# B&R Automation Studio project NAEUL004C00R13L518F00 (part 11)

#### Act_OptPage.st
```iecst
ACTION Act_OptPage:

	//Prevent Screen Saver Interupt Program
	IF tyProperty.tyVisu.uiCurrPage <> 0 THEN
		eCurrPage := tyProperty.tyVisu.uiCurrPage;
	ELSE
		Act_OptP0000McStatus;
		Act_OptP0000RunningNm;
		Act_OptP0000StatDisp;
	END_IF

	Act_OptP0000DisableSSaver;
	Act_OptP0000TouchTimer;			//Auto Logout
	Act_OptP0000Hermes; 	//Changed

	IF (tyProperty.tyVisu.uiChgPage = 65535) AND (usiChgPage = 0) THEN

		Act_OptC0005GoHomeCtrl;
		Act_OptC0005ShowNotif;
		Act_OptC0005AutoCtrl;
		Act_OptC0005RstErr;
		Act_OptC0005StatBarCtrl;
		Act_OptC0005Buzzer;
		Act_OptC0005ChgPage;
		Act_OptC0007Notif;
		Act_OptC0009Info;

		Act_OptP0202InsertRmvMag;
		Act_OptP0203InsertRmvMag;
		Act_OptP0204InsertRmvMag;

		CASE eCurrPage OF

			UIP0001Startup:
				Act_OptP0001Startup;

			UIP0100Login:
				Act_OptP0100Keypad;
				Act_OptP0100NomLogin;
				Act_OptP0100BypassLogin;
				Act_OptP0100Logout;

			UIP0200OpsGen:
				Act_OptP0200ChgPage;
				Act_OptP0200UpdtDat;
				Act_OptP0200VSMEMA;
				Act_OptP0200RcyMsg;
				Act_OptP0200ToP0204_P0003AccDat;
				Act_OptP0200ToP0204BypsInitConv;
				Act_OptP0202RstMnl;
				Act_OptP0203RstMnl;
				Act_OptP0204RstMnl;

			UIP0201OpsTravLifter:
				Act_OptP0201Navi;
				Act_OptP0201UpdtDat;
				Act_OptP0201IOMonitor;
				Act_OptP0201ChgParam;
				Act_OptP0200ToP0204_P0003AccDat;
				Act_OptP0200ToP0204BypsInitConv;
					//Changed
				Act_OptP0201QueryBoardInfo;
				Act_OptP0201CurrWorkOrderInfo;
				Act_OptP0201QueryWorkOrderInfo;
				Act_OptP0201BarcodeScanner;

			UIP0202OpsMag1:
				Act_OptP0202Navi;
				Act_OptP0202UpdtDat;
				Act_OptP0202IOMonitor;
				Act_OptP0202ChgPage;
				Act_OptP0202_P0003AIVDat;
				Act_OptP0202ChgParam;
				Act_OptP0200ToP0204_P0003AccDat;
				Act_OptP0200ToP0204BypsInitConv;
				Act_OptP0202ToP0204_P0003UnloadMag;
				IF p_tyNtParamCurr.bProjMagConvLane1Prep THEN
					Act_OptP0202Lane1ChgMag;
				END_IF
			UIP0203OpsMag2:
				Act_OptP0203Navi;
				Act_OptP0203UpdtDat;
				Act_OptP0203IOMonitor;
				Act_OptP0203ChgPage;
				Act_OptP0203_P0003AIVDat;
				Act_OptP0203ChgParam;
				Act_OptP0200ToP0204_P0003AccDat;
				Act_OptP0200ToP0204BypsInitConv;
				Act_OptP0202ToP0204_P0003UnloadMag;
				IF p_tyNtParamCurr.bProjMagConvLane2Prep THEN
					Act_OptP0203Lane2ChgMag;
				END_IF
			UIP0204OpsMag3:
				Act_OptP0204Navi;
				Act_OptP0204UpdtDat;
				Act_OptP0204IOMonitor;
				Act_OptP0204ChgPage;
				Act_OptP0204_P0003AIVDat;
				Act_OptP0204ChgParam;
				Act_OptP0200ToP0204_P0003AccDat;
				Act_OptP0200ToP0204BypsInitConv;
				Act_OptP0202ToP0204_P0003UnloadMag;

			UIP0205OpsAIV:
				Act_OptP0205Navi;
				Act_OptP0205IOMonitor;

			UIP0206OpsMagConv1:
				Act_OptP0206Navi;
				Act_OptP0206UpdtDat;
				Act_OptP0206IOMonitor;
				Act_OptP0200ToP0204_P0003AccDat;
				Act_OptP0200ToP0204BypsInitConv;

			UIP0207OpsMagConv2:
				Act_OptP0207Navi;
				Act_OptP0207UpdtDat;
				Act_OptP0207IOMonitor;
				Act_OptP0200ToP0204_P0003AccDat;
				Act_OptP0200ToP0204BypsInitConv;

			UIP0300McInfo:

			UIP0400ProdSel:
				Act_OptP0400Search;
				Act_OptP0400Load;
				Act_OptP0400Preview;
				Act_OptP0400Table;
				Act_OptP0400Keypad;
				Act_OptP0400Mask;
				Act_OptP0400Sort;
				Act_OptP0400RcpPopUp;

			UIP0410MagSel:
				Act_OptP0410Load;
				Act_OptP0410Preview;
				Act_OptP0410Table;
				Act_OptP0410Mask;
				Act_OptP0410Sort;

			UIP0600Alm:
				Act_OptP0600Alm;
				Act_OptP0600RcyMsg;

			UIP0700LFCtrl:
				Act_OptP0700LFLeaderCtrl;
				Act_OptP0700Mask;
				Act_OptP0700Table;

			UIP0800MagInfo:
				Act_OptP0800Table1;
				Act_OptP0800Mag1Updt;
				Act_OptP0800Table2;
				Act_OptP0800Mag2Updt;
				Act_OptP0800Table3;
				Act_OptP0800Mag3Updt;

			UIP0850OvenInfo:
				Act_OptP0850UpdtDat;
				Act_OptP0850BrdInOven;
				Act_OptP0850Keypad;

				UIP0002Menu,UIP0003MMenu, UIP0900GenIn, UIP0910GenOut, UIP0920MtrNPneuCtrl, UIP0921Shutter, UIP0922Stopper, UIP0923SafetyBar, UIP0926LifterConv, UIP0927LifterConv2, UIP0928MagConv, UIP0929MagConv2,UIP0930MagConv1, UIP0931MagConv2, UIP0932MagConv3, UIP0933PusherConv,
				 UIP0934AW, UIP0935Lifter, UIP0936Trav, UIP0937AWPushOrPuller, UIP0938MagAW, UIP0939Lifter2,UIP0940CommCtrl:
				IF eCurrPage = UIP0002Menu THEN
					Act_OptP0002Mask;
					Act_OptP0002ChgPage;
					Act_OptP0002MsgGuide;
					Act_OptP0002UpdtData;
				END_IF

				IF eCurrPage = UIP0003MMenu THEN
					Act_OptP0003UpdtStat;
					Act_OptP0202ToP0204_P0003UnloadMag;
					Act_OptP0200ToP0204_P0003AccDat;
					Act_OptP0202_P0003AIVDat;
					Act_OptP0203_P0003AIVDat;
					Act_OptP0204_P0003AIVDat;
				END_IF

				Act_OptP0002ManualCtrl;
				Act_OptP0910RstMnl;
				Act_OptP0921RstMnl;
				Act_OptP0922RstMnl;
				Act_OptP0923RstMnl;
				IF p_tyNtParamCurr.bProjMagConvLane1Prep THEN
					Act_OptP0926RstMnl;
					Act_OptP0928RstMnlTop;
					Act_OptP0928RstMnlBtm;
				END_IF
				IF p_tyNtParamCurr.bProjMagConvLane2Prep THEN
					Act_OptP0927RstMnl;
					Act_OptP0929RstMnlTop;
					Act_OptP0929RstMnlBtm;
				END_IF
				Act_OptP0930RstMnl;
				Act_OptP0931RstMnl;
				Act_OptP0932RstMnl;
				Act_OptP0933RstMnl;
				Act_OptP0934RstMnl;
				Act_OptP0935RstMnl;
				Act_OptP0936RstMnl;
				Act_OptP0937RstMnl;
				Act_OptP0938RstMnl;
				IF p_tyNtParamCurr.bProjLifter2Prep THEN
					Act_OptP0939RstMnl;
				END_IF
				Act_OptP0940RstMnl;
				Act_OptP0950RstMnl;
				Act_OptP0202RstMnl;
				Act_OptP0203RstMnl;
				Act_OptP0204RstMnl;
				Act_OptP0205RstMnl;

				IF bUIManualMod = TRUE THEN

					//General Input
					Act_OptP0900ReadDI;

					//General Output
					Act_OptP0910WriteDO;

					//MtrNPneuCtrl
					Act_OptP0920FullMask;
					Act_OptP0920ChgPage;

					//Inlet & Outlet Shutter
					Act_OptP0921DualMask;
					Act_OptP0921Navi;
					Act_OptP0921InletShutterChgLyr;
					Act_OptP0921InletShutterSen;
					Act_OptP0921InletShutterFB;
					Act_OptP0921InletShutterFBStat;
					Act_OptP0921InletShutterDC;
					Act_OptP0921OutletShutterChgLyr;
					Act_OptP0921OutletShutterSen;
					Act_OptP0921OutletShutterFB;
					Act_OptP0921OutletShutterFBStat;
					Act_OptP0921OutletShutterDC;
					Act_OptP0921OutletShutterChgLyr2;
					Act_OptP0921OutletShutterSen2;
					Act_OptP0921OutletShutterFB2;
					Act_OptP0921OutletShutterFBStat2;
					Act_OptP0921OutletShutterDC2;
					Act_OptP0921OutletShutterChgLyr3;
					Act_OptP0921OutletShutterSen3;
					Act_OptP0921OutletShutterFB3;
					Act_OptP0921OutletShutterFBStat3;
					Act_OptP0921OutletShutterDC3;

					//Stopper A & B
					Act_OptP0922DualMask;
					Act_OptP0922Navi;
					Act_OptP0922StopperAChgLyr;
					Act_OptP0922StopperASen;
					Act_OptP0922StopperAFB;
					Act_OptP0922StopperAFBStat;
					Act_OptP0922StopperADC;
					Act_OptP0922StopperBChgLyr;
					Act_OptP0922StopperBSen;
					Act_OptP0922StopperBFB;
					Act_OptP0922StopperBFBStat;
					Act_OptP0922StopperBDC;
					Act_OptP0922InStopperChgLyr;
					Act_OptP0922InStopperSen;
					Act_OptP0922InStopperFB;
					Act_OptP0922InStopperFBStat;
					Act_OptP0922InStopperDC;

					//Safety Bar
					Act_OptP0923DualMask;
					Act_OptP0923Navi;
					Act_OptP0923Mag1SafetyBarChgLyr;
					Act_OptP0923Mag1SafetyBarSen;
					Act_OptP0923Mag1SafetyBarFB;
					Act_OptP0923Mag1SafetyBarFBStat;
					Act_OptP0923Mag1SafetyBarDC;
					Act_OptP0923Mag2SafetyBarChgLyr;
					Act_OptP0923Mag2SafetyBarSen;
					Act_OptP0923Mag2SafetyBarFB;
					Act_OptP0923Mag2SafetyBarFBStat;
					Act_OptP0923Mag2SafetyBarDC;
					Act_OptP0923Mag3SafetyBarChgLyr;
					Act_OptP0923Mag3SafetyBarSen;
					Act_OptP0923Mag3SafetyBarFB;
					Act_OptP0923Mag3SafetyBarFBStat;
					Act_OptP0923Mag3SafetyBarDC;

					IF p_tyNtParamCurr.bProjMagConvLane1Prep  THEN
						//Lifter Magazine Conveyor
						Act_OptP0926FullMask;
						Act_OptP0926Navi;
						Act_OptP0926LifterMagConvChgLyr;
						Act_OptP0926LifterMagConvSen;
						Act_OptP0926LifterMagConvFB;
						Act_OptP0926LifterMagConvFBStat;
						Act_OptP0926LifterMagConvDC;

						//MagConv Lane1
						Act_OptP0928FullMask;
						Act_OptP0928Navi;
						Act_OptP0928MagConv1ChgLyr;
						Act_OptP0928MagConv1Sen;
						Act_OptP0928MagConv1TopFB;
						Act_OptP0928MagConv1BtmFB;
						Act_OptP0928MagConv1FBStat;
						Act_OptP0928MagConv1TopDC;
						Act_OptP0928MagConv1BtmDC;
					END_IF

					IF p_tyNtParamCurr.bProjMagConvLane2Prep  THEN
						//Lifter Magazine Conveyor2
						Act_OptP0927FullMask;
						Act_OptP0927Navi;
						Act_OptP0927LifterMagConvChgLyr;
						Act_OptP0927LifterMagConvSen;
						Act_OptP0927LifterMagConvFB;
						Act_OptP0927LifterMagConvFBStat;
						Act_OptP0927LifterMagConvDC;

						//MagConv Lane2
						Act_OptP0929FullMask;
						Act_OptP0929Navi;
						Act_OptP0929MagConv2ChgLyr;
						Act_OptP0929MagConv2Sen;
						Act_OptP0929MagConv2TopFB;
						Act_OptP0929MagConv2BtmFB;
						Act_OptP0929MagConv2FBStat;
						Act_OptP0929MagConv2TopDC;
						Act_OptP0929MagConv2BtmDC;
					END_IF

					//Magazine Conveyor 1
					Act_OptP0930FullMask;
					Act_OptP0930Navi;
					Act_OptP0930MagConv1ChgLyr;
					Act_OptP0930MagConv1Sen;
					Act_OptP0930MagConv1FB;
					Act_OptP0930MagConv1FBStat;
					Act_OptP0930MagConv1DC;

					//Magazine Conveyor 2
					Act_OptP0931FullMask;
					Act_OptP0931Navi;
					Act_OptP0931MagConv2ChgLyr;
					Act_OptP0931MagConv2Sen;
					Act_OptP0931MagConv2FB;
					Act_OptP0931MagConv2FBStat;
					Act_OptP0931MagConv2DC;

					//Magazine Conveyor 3
					Act_OptP0932FullMask;
					Act_OptP0932Navi;
					Act_OptP0932MagConv3ChgLyr;
					Act_OptP0932MagConv3Sen;
					Act_OptP0932MagConv3FB;
					Act_OptP0932MagConv3FBStat;
					Act_OptP0932MagConv3DC;

					//Pusher Conveyor
					Act_OptP0933FullMask;
					Act_OptP0933Navi;
					Act_OptP0933PusherConvChgLyr;
					Act_OptP0933PusherConvSen;
					Act_OptP0933PusherConvFB;
					Act_OptP0933PusherConvFBStat;
					Act_OptP0933PusherConvDC;

					//AutoWidth
					Act_OptP0934FullMask;
					Act_OptP0934Navi;
					Act_OptP0934FBCtrl;
					Act_OptP0934FBStat;
					Act_OptP0934Mask;
					Act_OptP0934UpdtDat;
					Act_OptP0934Keypad;

					//Lifter
					Act_OptP0935FullMask;
					Act_OptP0935Navi;
					Act_OptP0935FBCtrl;
					Act_OptP0935FBStat;
					Act_OptP0935Mask;
					Act_OptP0935UpdtDat;
					Act_OptP0935Keypad;

					//Traverser
					Act_OptP0936FullMask;
					Act_OptP0936Navi;
					Act_OptP0936FBCtrl;
					Act_OptP0936FBStat;
					Act_OptP0936Mask;
					Act_OptP0936UpdtDat;
					Act_OptP0936Keypad;

					//Pusher Or Puller Auto Width
					Act_OptP0937FullMask;
					Act_OptP0937Navi;
					Act_OptP0937FBCtrl;
					Act_OptP0937FBStat;
					Act_OptP0937Mask;
					Act_OptP0937UpdtDat;
					Act_OptP0937Keypad;

					//Magazine Auto Width
					Act_OptP0938FullMask;
					Act_OptP0938Navi;
					Act_OptP0938FBCtrl1;
					Act_OptP0938FBCtrl2;
					Act_OptP0938FBCtrl3;
					Act_OptP0938FBStat;
					Act_OptP0938Mask;
					Act_OptP0938UpdtDat;
					Act_OptP0938Keypad;

					//Lifter 2
					IF p_tyNtParamCurr.bProjLifter2Prep THEN
						Act_OptP0939FullMask;
						Act_OptP0939Navi;
						Act_OptP0939FBCtrl;
						Act_OptP0939FBStat;
						Act_OptP0939Mask;
						Act_OptP0939UpdtDat;
						Act_OptP0939Keypad;
					END_IF
					//Communication
					Act_OptP0940FullMask;
					Act_OptP0940ReadDI;
					Act_OptP0940WriteDO;

				END_IF

			UIP0950Simu:
				Act_OptP0950Navi;
				Act_OptP0950Ctrl;
				Act_OptP0950SimuMod;
				//Act_OptP0950DispBffrCycle;

			UIP1000Lang:
				Act_OptP1000SelectLang;
				Act_OptP1000Keypad;

			UIP1020McSetNavi:
				Act_OptP1020Navi;

			UIP1021McSetGen:
				Act_OptP1021Navi;
				Act_OptP1021Save;
				Act_OptP1021Keypad;
				Act_OptP1021Teach;
				Act_OptP1021IPAddr;
				Act_OptP1021SubnetMask;
				Act_OptP1021HMIIPAddr;
				Act_OptP1021DHCPSetting;

			UIP1022McSetVComm:
				Act_OptP1022Navi;
				Act_OptP1022Save;
				Act_OptP1022DisLF;
				Act_OptP1022Keypad; //new for Hermes 1.3

			UIP1023McSetHComm:
				Act_OptP1023Navi;
				Act_OptP1023ShowLyr;
				Act_OptP1023Save;
				Act_OptP1023USSel;
				Act_OptP1023Keypad;

			UIP1024McSetAntiGap:
				Act_OptP1024Navi;
				Act_OptP1024Save;
				Act_OptP1024Keypad;

			UIP1025McSetScan:
				Act_OptP1025Navi;
				Act_OptP1025Save;
				Act_OptP1025Keypad;

			UIP1026McSetTeach:
				Act_OptP1026Navi;
				Act_OptP1026FullMask;
				Act_OptP1026Mnl;

				//Traverser
				Act_OptP1026TravTeach;
				Act_OptP1026TravFBCtrl;
				Act_OptP1026TravFBStat;
				Act_OptP1026TravMask;
				Act_OptP1026TravUpdtDat;
				Act_OptP1026TravKeypad;
				Act_OptP1026TravRstMnl;

				//Lifter
				Act_OptP1026LifterTeach;
				IF (bTeachLifterTopPos2 OR bTeachLifterBtmPos2) AND  p_tyNtParamCurr.bProjLifter2Prep THEN
					Act_OptP1026Lifter2FBCtrl;
					Act_OptP1026Lifter2FBStat;
					Act_OptP1026Lifter2Mask;
					Act_OptP1026Lifter2UpdtDat;
				ELSE
					Act_OptP1026LifterFBCtrl;
					Act_OptP1026LifterFBStat;
					Act_OptP1026LifterMask;
					Act_OptP1026LifterUpdtDat;
				END_IF
				Act_OptP1026LifterKeypad;
				Act_OptP1026LifterRstMnl;

			UIP1027McSetOpCon:
				Act_OptP1027Navi;
				Act_OptP1027Save;
				Act_OptP1027Keypad;

			UIP1030MagSet:
				Act_OptP1030Mask;
				Act_OptP1030Save;
				Act_OptP1030Del;
				Act_OptP1030Table;
				Act_OptP1030LoadData;
				Act_OptP1030Keypad;
				Act_OptP1030Teach;
				Act_OptP1030Sort;

			UIP1031MagSetTeach:
				Act_OptP1031Navi;
				Act_OptP1031FullMask;
				Act_OptP1031Mnl;

				//Traverser
				Act_OptP1031TravTeach;
				Act_OptP1031TravFBCtrl;
				Act_OptP1031TravFBStat;
				Act_OptP1031TravMask;
				Act_OptP1031TravUpdtDat;
				Act_OptP1031TravKeypad;
				Act_OptP1031TravRstMnl;

				//Lifter
				Act_OptP1031LifterTeach;

				IF p_tyNtParamCurr.bProjMagConvLane2Prep AND bTeachLifterMag2Slt1Pos AND  p_tyNtParamCurr.bProjLifter2Prep THEN
					Act_OptP1031Lifter2FBCtrl;
					Act_OptP1031Lifter2FBStat;
					Act_OptP1031Lifter2Mask;
					Act_OptP1031Lifter2UpdtDat;
				ELSE
					Act_OptP1031LifterFBCtrl;
					Act_OptP1031LifterFBStat;
					Act_OptP1031LifterMask;
					Act_OptP1031LifterUpdtDat;
				END_IF
				Act_OptP1031LifterKeypad;
				Act_OptP1031LifterRstMnl;

			UIP1040ProdSet:
				Act_OptP1040Mask;
				Act_OptP1040Save;
				Act_OptP1040Limit;
				Act_OptP1040Del;
				Act_OptP1040Table;
				Act_OptP1040LoadData;
				Act_OptP1040Search;
				Act_OptP1040Keypad;
				Act_OptP1040ToXML;
				Act_OptP1040FromXML;
				Act_OptP1040Sort;
				Act_OptP1040RcpPopUp;

			UIP1050LFSet:
				Act_OptP1050Keypad;
				Act_OptP1050Edit;
				Act_OptP1050Online;
				Act_OptP1050Offline;
				Act_OptP1050Delete;
				Act_OptP1050ShftUp;
				Act_OptP1050ShftDwn;
				Act_OptP1050Mask;
				Act_OptP1050Table;
				Act_OptP1050Oven;

			UIP1080UsrMgmt:
				Act_OptP1080Keypad;
				Act_OptP1080AddUsr;
				Act_OptP1080DelUsr;
				Act_OptP1080EditUsr;
				Act_OptP1080EditAccess;
				Act_OptP1080Table;

			UIP1081UsrMgmtUsrAccessRgt:
				Act_OptP1081Navi;
				Act_OptP1081Save;
				Act_OptP1081Load;
				Act_OptP1081Keypad;

		END_CASE

	END_IF

END_ACTION
```

#### Act_OptC0005GoHomeCtrl.st
```iecst
ACTION Act_OptC0005GoHomeCtrl:

	//Control
	IF tyCommon.tyMain.tyBtnHome.bRtCompl = TRUE OR tyCommon.tyMain1.tyBtnHome.bRtCompl = TRUE THEN
		tyCommon.tyMain.tyBtnHome.bRtCompl	:= FALSE;
		tyCommon.tyMain1.tyBtnHome.bRtCompl := FALSE;
		eChgPage							:= UIP0002Menu;
	END_IF

	//Go Main
	IF tyCommon.tyMain.tyBtnGoMain.bRtCompl = TRUE THEN
		tyCommon.tyMain.tyBtnGoMain.bRtCompl := FALSE;
		eChgPage		:= UIP0003MMenu;
	END_IF

	//Mask
	IF tyP0100Login.tyLogin.tyBtnLogin.bRtCompl 					OR tyP0100Login.tyLogout.tyBtnLogout.bRtCompl
		OR tyP0400ProdSel.tyProdSel.tyBtnLoad.bRtCompl 				OR tyP0400ProdSel.tyProdSel.tyStringSearch.bRtCompl
		OR tyP0410MagSel.tyMagSel.tyBtnLoad.bRtCompl				OR tyP0800MagInfo.tyMagInfo1.tyBtnMag1SetFull.bRtCompl
		OR tyP0800MagInfo.tyMagInfo1.tyBtnMag2SetFull.bRtCompl		OR tyP0800MagInfo.tyMagInfo2.tyBtnMag3SetFull.bRtCompl
		OR tyP1030MagSet.tyMagSet.tyBtnDelete.bRtCompl				OR tyP1030MagSet.tyMagSet.tyBtnSave.bRtCompl
		OR tyP1040ProdSet.tyProdSet.tyBtnDelete.bRtCompl			OR tyP1040ProdSet.tyProdSet.tyBtnSave.bRtCompl
		OR tyP1040ProdSet.tyProdSet.tyBtnToXML.bRtCompl				OR tyP1040ProdSet.tyProdSet.tyBtnFromXML.bRtCompl
		OR tyP1050LFSet.tyLdr.tyBtnDelete.bRtCompl					OR tyP1050LFSet.tyLdr.tyBtnOnline.bRtCompl
		OR tyP1050LFSet.tyLdr.tyBtnOffline.bRtCompl					OR tyP1050LFSet.tyLdr.tyBtnShftUp.bRtCompl
		OR tyP1050LFSet.tyLdr.tyBtnShftDwn.bRtCompl					OR tyP1080UsrMgmt.tyUsrMgmt.tyBtnDeleteUsr.bRtCompl
		OR tyP1080UsrMgmt.tyUsrMgmt.tyBtnEditDetail.bRtCompl		OR tyP1080UsrMgmt.tyUsrMgmt.tyBtnNewUsr.bRtCompl
		OR tyCommon.tySet.tyBtnSave.bRtCompl						OR bTeachTravPosA
		OR bTeachTravPosB											OR bTeachTravPosMag1
		OR bTeachTravPosMag2										OR bTeachTravPosMag3
		OR bTeachLifterPosA											OR bTeachLifterPosB
		OR bTeachLifterMag1Slt1Pos									OR bTeachLifterMag2Slt1Pos
		OR bTeachLifterMag3Slt1Pos
		OR p_bSimuStatusRun
		THEN

		fUIInRtStatOff(ADR(tyCommon.tyMain.tyBtnHome.uiMaskRtStat));
		fUIInRtStatOff(ADR(tyCommon.tyMain1.tyBtnHome.uiMaskRtStat));

		fUIInRtStatOff(ADR(tyCommon.tyMain.tyBtnGoMain.uiMaskRtStat));

	ELSIF bUIManualMod THEN
		fUIInRtStatHide(ADR(tyCommon.tyMain.tyBtnHome.uiMaskRtStat));
		fUIInRtStatHide(ADR(tyCommon.tyMain1.tyBtnHome.uiMaskRtStat));

		fUIInRtStatHide(ADR(tyCommon.tyMain.tyBtnGoMain.uiMaskRtStat));
	ELSE
		fUIInRtStatHide(ADR(tyCommon.tyMain.tyBtnHome.uiMaskRtStat));
		fUIInRtStatHide(ADR(tyCommon.tyMain1.tyBtnHome.uiMaskRtStat));

		fUIInRtStatHide(ADR(tyCommon.tyMain.tyBtnGoMain.uiMaskRtStat));
	END_IF

END_ACTION
```

#### Act_OptC0005ShowNotif.st
```iecst
ACTION Act_OptC0005ShowNotif:

	//Control
	IF tyCommon.tyMain.tyBtnNotification.bRtCompl = TRUE OR tyCommon.tyMain1.tyBtnNotification.bRtCompl = TRUE THEN
		tyCommon.tyMain.tyBtnNotification.bRtCompl		:= FALSE;
		tyCommon.tyMain1.tyBtnNotification.bRtCompl		:= FALSE;

		fUIInRtStatOff(ADR(tyCommon.tyNotif.tyLyr.uiRtStat));
	END_IF

END_ACTION
```

#### Act_OptC0005RstErr.st
```iecst
ACTION Act_OptC0005RstErr:

	//Control
	IF tyCommon.tyMain.tyBtnReset.bRtCompl = TRUE OR tyP0003MMenu.tyMMenuBtn.tyBtnReset.bRtCompl = TRUE THEN
		eRstErrAct	:= RstErrActRun;

		IF NOT p_tyDI.bCurtainSafetySig THEN
			bSafetyCurtainReset := TRUE;//Curtain reset button //Update For Curtain Sensor
		END_IF

//		fbCurtainRstDly(IN:= TRUE);

		IF p_eRstErrStat = RstErrActRun AND p_eRstErrStatus =  Done THEN
			eRstErrAct	:= RstErrActIdle;

			tyCommon.tyMain.tyBtnReset.bRtCompl	:= FALSE;

			tyP0003MMenu.tyMMenuBtn.tyBtnReset.bRtCompl := FALSE;
		END_IF

	END_IF

	//Mask
	IF p_bAlarmErr = TRUE OR p_bAlarmWarning = TRUE OR p_tyDI.bSafetyRlySig = FALSE THEN
		fUIInRtStatHide(ADR(tyCommon.tyMain.tyBtnReset.uiMaskRtStat));

		fUIInRtStatHide(ADR(tyP0003MMenu.tyMMenuBtn.tyBtnStop.uiRtStat));
		fUIInRtStatHide(ADR(tyP0003MMenu.tyMMenuBtn.tyBtnStop.uiMaskRtStat));

	ELSE
		fUIInRtStatOff(ADR(tyCommon.tyMain.tyBtnReset.uiMaskRtStat));
		fUIInRtStatOff(ADR(tyP0003MMenu.tyMMenuBtn.tyBtnStop.uiRtStat));
	END_IF

//	fbCurtainRstDly (IN := bSafetyCurtainReset);
//	IF fbCurtainRstDly.Q THEN
//		bSafetyCurtainReset := FALSE;
//	END_IF

	IF bSafetyCurtainReset THEN
		fbCurtainRstDly(IN:=TRUE);

		IF fbCurtainRstDly.Q THEN
			fbCurtainRstDly(IN:= FALSE);
			bSafetyCurtainReset := FALSE;
		END_IF
	END_IF

END_ACTION
```

#### Act_OptC0005Buzzer.st
```iecst
ACTION Act_OptC0005Buzzer:

	IF tyCommon.tyMain.tyBtnBuzzer.bRtCompl = TRUE OR tyP0003MMenu.tyMMenuBtn.tyBtnBuz.bRtCompl = TRUE THEN
		tyCommon.tyMain.tyBtnBuzzer.bRtCompl		:= FALSE;
		tyP0003MMenu.tyMMenuBtn.tyBtnBuz.bRtCompl	:= FALSE;

		IF eCurrPage = UIP0003MMenu THEN
			tyCommon.tyMain.tyBtnBuzzer.bValue		:= tyP0003MMenu.tyMMenuBtn.tyBtnBuz.bValue;
		ELSE
			tyP0003MMenu.tyMMenuBtn.tyBtnBuz.bValue 	:=  tyCommon.tyMain.tyBtnBuzzer.bValue;
		END_IF

		IF tyCommon.tyMain.tyBtnBuzzer.bValue = TRUE OR tyP0003MMenu.tyMMenuBtn.tyBtnBuz.bValue = TRUE THEN
			tyCommon.tyMain.tyBtnBuzzer.usiBitmapIdx		:= 2;
			tyP0003MMenu.tyMMenuBtn.tyBtnBuz.usiBitmapIdx 	:= 2;

			bMuteBuz	:= TRUE;
		ELSE
			tyCommon.tyMain.tyBtnBuzzer.usiBitmapIdx		:= 1;
			tyP0003MMenu.tyMMenuBtn.tyBtnBuz.usiBitmapIdx 	:= 1;

			bMuteBuz	:= FALSE;
		END_IF

	END_IF

	//Mute Buzzer
	IF EDGEPOS((p_bAlarmErr OR p_bAlarmWarning OR p_bAlarmInfo) (*AND NOT bUIManualMod*)) THEN

		tyCommon.tyMain.tyBtnBuzzer.bValue				:= FALSE;
		tyCommon.tyMain.tyBtnBuzzer.bRtLk				:= FALSE;
		tyCommon.tyMain.tyBtnBuzzer.usiBitmapIdx		:= 1;

		tyP0003MMenu.tyMMenuBtn.tyBtnBuz.bValue 		:= FALSE;
		tyP0003MMenu.tyMMenuBtn.tyBtnBuz.usiBitmapIdx 	:= 1;

		bMuteBuz	:= FALSE;

	ELSIF (p_bAlarmErr OR p_bAlarmWarning OR p_bAlarmInfo) THEN

		IF p_bAlarmInfoLF AND NOT (p_bAlarmErr OR p_bAlarmWarning OR (p_bAlarmInfo AND NOT p_bAlarmInfoLF)) THEN

			IF p_tyMcParamCurr.bLFBuzMute THEN

				tyCommon.tyMain.tyBtnBuzzer.bValue				:= FALSE;
				tyCommon.tyMain.tyBtnBuzzer.bRtLk				:= TRUE;
				tyCommon.tyMain.tyBtnBuzzer.usiBitmapIdx		:= 0;

				tyP0003MMenu.tyMMenuBtn.tyBtnBuz.bValue 		:= FALSE;
				tyP0003MMenu.tyMMenuBtn.tyBtnBuz.usiBitmapIdx 	:= 0;

				bMuteBuz	:= FALSE;
			ELSE
				tyCommon.tyMain.tyBtnBuzzer.bRtLk				:= FALSE;

				IF tyCommon.tyMain.tyBtnBuzzer.bValue OR tyP0003MMenu.tyMMenuBtn.tyBtnBuz.bValue THEN
					tyCommon.tyMain.tyBtnBuzzer.usiBitmapIdx		:= 2;

					tyP0003MMenu.tyMMenuBtn.tyBtnBuz.usiBitmapIdx   := 2;
				ELSE
					tyCommon.tyMain.tyBtnBuzzer.usiBitmapIdx		:= 1;

					tyP0003MMenu.tyMMenuBtn.tyBtnBuz.usiBitmapIdx   := 1;
				END_IF

			END_IF
		ELSE

			tyCommon.tyMain.tyBtnBuzzer.bRtLk				:= FALSE;

			IF tyCommon.tyMain.tyBtnBuzzer.bValue OR tyP0003MMenu.tyMMenuBtn.tyBtnBuz.bValue THEN
				tyCommon.tyMain.tyBtnBuzzer.usiBitmapIdx		:= 2;

				tyP0003MMenu.tyMMenuBtn.tyBtnBuz.usiBitmapIdx   := 2;
			ELSE
				tyCommon.tyMain.tyBtnBuzzer.usiBitmapIdx		:= 1;

				tyP0003MMenu.tyMMenuBtn.tyBtnBuz.usiBitmapIdx   := 1;
			END_IF
		END_IF

	ELSIF NOT(p_bAlarmErr OR p_bAlarmWarning OR p_bAlarmInfo) (*OR bUIManualMod*) THEN
		tyCommon.tyMain.tyBtnBuzzer.bRtLk				:= TRUE;
		tyCommon.tyMain.tyBtnBuzzer.usiBitmapIdx		:= 0;

		tyP0003MMenu.tyMMenuBtn.tyBtnBuz.usiBitmapIdx   := 0;

		bMuteBuz	:= FALSE;
	END_IF

END_ACTION
```

#### Act_OptC0005AutoCtrl.st
```iecst
ACTION Act_OptC0005AutoCtrl:

	//Control
	//Error
	IF EDGEPOS(p_bAlarmErr = TRUE AND p_bOpsStatusStop = FALSE) THEN

		tyCommon.tyMain.tyBtnStart.bRtCompl	:= FALSE;
		tyCommon.tyMain.tyBtnStop.bRtCompl	:= FALSE;
		tyCommon.tyMain.tyBtnStep.bRtCompl	:= FALSE;

		tyCommon.tyMain.tyBtnStart.bValue	:= FALSE;
		tyCommon.tyMain.tyBtnStop.bValue	:= FALSE;
		tyCommon.tyMain.tyBtnStep.bValue	:= FALSE;

		//Additional HMI Control

		tyP0003MMenu.tyMMenuBtn.tyBtnAuto.bRtCompl  := FALSE;
		tyP0003MMenu.tyMMenuBtn.tyBtnStop.bRtCompl  := FALSE;

		tyP0003MMenu.tyMMenuBtn.tyBtnAuto.bValue 	:= FALSE;
		tyP0003MMenu.tyMMenuBtn.tyBtnStop.bValue 	:= FALSE;

		eOpsAct	:= OperationsActError;

	ELSE

		IF p_eOpsStat = OperationsActError AND p_eOpsStatus = Done THEN
			eOpsAct	:= OperationsActIdle;
		END_IF

	END_IF

	//Start
	IF tyCommon.tyMain.tyBtnStart.bRtCompl = TRUE OR tyP0003MMenu.tyMMenuBtn.tyBtnAuto.bRtCompl  THEN

		IF tyCommon.tyMain.tyBtnStart.bValue = TRUE OR tyP0003MMenu.tyMMenuBtn.tyBtnAuto.bValue = TRUE  THEN

			IF eCurrPage <> UIP0200OpsGen AND eCurrPage <> UIP0201OpsTravLifter AND eCurrPage <> UIP0202OpsMag1 AND eCurrPage <> UIP0203OpsMag2 AND eCurrPage <> UIP0204OpsMag3
				AND NOT tyP0003MMenu.tyMMenuBtn.tyBtnAuto.bValue THEN

				IF bChgPage = FALSE THEN
					bChgPage	:= TRUE;
					eChgPage	:= UIP0200OpsGen;
				ELSE
					IF eChgPage <> UIP0200OpsGen THEN
						bChgPage	:= FALSE;

						tyCommon.tyMain.tyBtnStart.bRtCompl	:= FALSE;
						tyCommon.tyMain.tyBtnStart.bValue	:= FALSE;
					END_IF
				END_IF

			ELSE
				bChgPage	:= FALSE;

				tyCommon.tyMain.tyBtnStart.bValue	:= FALSE;

				tyCommon.tyMain.tyBtnStop.bRtCompl	:= FALSE;
				tyCommon.tyMain.tyBtnStep.bRtCompl	:= FALSE;

				tyCommon.tyMain.tyBtnStop.bValue	:= FALSE;
				tyCommon.tyMain.tyBtnStep.bValue	:= FALSE;

				tyP0003MMenu.tyMMenuBtn.tyBtnAuto.bValue := FALSE;

				tyP0003MMenu.tyMMenuBtn.tyBtnStop.bRtCompl := FALSE;
				tyP0003MMenu.tyMMenuBtn.tyBtnStop.bValue   := FALSE;

			END_IF

		ELSE

			eOpsAct	:= OperationsActStart;

			IF p_eOpsStat = OperationsActStart AND p_eOpsStatus = Done THEN
				eOpsAct	:= OperationsActIdle;

				tyCommon.tyMain.tyBtnStart.bRtCompl		   := FALSE;
				tyP0003MMenu.tyMMenuBtn.tyBtnAuto.bRtCompl := FALSE;

			END_IF

		END_IF

	END_IF

	//Stop
	IF tyCommon.tyMain.tyBtnStop.bRtCompl = TRUE OR tyP0003MMenu.tyMMenuBtn.tyBtnStop.bRtCompl  THEN

		IF tyCommon.tyMain.tyBtnStop.bValue = TRUE OR tyP0003MMenu.tyMMenuBtn.tyBtnStop.bValue THEN

			tyCommon.tyMain.tyBtnStop.bValue			:= FALSE;
			tyP0003MMenu.tyMMenuBtn.tyBtnStop.bValue	:= FALSE;

			tyCommon.tyMain.tyBtnStart.bRtCompl	:= FALSE;
			tyCommon.tyMain.tyBtnStep.bRtCompl	:= FALSE;

			tyP0003MMenu.tyMMenuBtn.tyBtnAuto.bRtCompl	:= FALSE;

			tyCommon.tyMain.tyBtnStart.bValue	:= FALSE;
			tyCommon.tyMain.tyBtnStep.bValue	:= FALSE;

			tyP0003MMenu.tyMMenuBtn.tyBtnAuto.bValue	:= FALSE;

		ELSE

			eOpsAct	:= OperationsActStop;

			IF p_eOpsStat = OperationsActStop AND p_eOpsStatus = Done THEN
				eOpsAct	:= OperationsActIdle;

				tyCommon.tyMain.tyBtnStop.bRtCompl	:= FALSE;

				tyP0003MMenu.tyMMenuBtn.tyBtnStop.bRtCompl	:= FALSE;
			END_IF

		END_IF

	END_IF

	//Step
	IF tyCommon.tyMain.tyBtnStep.bRtCompl = TRUE THEN

		IF tyCommon.tyMain.tyBtnStep.bValue = TRUE THEN

			IF eCurrPage <> UIP0200OpsGen AND eCurrPage <> UIP0201OpsTravLifter AND eCurrPage <> UIP0202OpsMag1 AND eCurrPage <> UIP0203OpsMag2 AND eCurrPage <> UIP0204OpsMag3 THEN

				IF bChgPage = FALSE THEN
					bChgPage	:= TRUE;
					eChgPage	:= UIP0200OpsGen;
				ELSE
					IF eChgPage <> UIP0200OpsGen THEN
						bChgPage	:= FALSE;

						tyCommon.tyMain.tyBtnStep.bRtCompl	:= FALSE;
						tyCommon.tyMain.tyBtnStep.bValue	:= FALSE;
					END_IF
				END_IF

			ELSE
				bChgPage	:= FALSE;

				tyCommon.tyMain.tyBtnStep.bValue	:= FALSE;

				tyCommon.tyMain.tyBtnStart.bRtCompl	:= FALSE;
				tyCommon.tyMain.tyBtnStop.bRtCompl	:= FALSE;

				tyCommon.tyMain.tyBtnStart.bValue	:= FALSE;
				tyCommon.tyMain.tyBtnStop.bValue	:= FALSE;
			END_IF

		ELSE

			eOpsAct	:= OperationsActStep;

			IF p_eOpsStat = OperationsActStep AND p_eOpsStatus = Done THEN
				eOpsAct	:= OperationsActIdle;

				tyCommon.tyMain.tyBtnStep.bRtCompl	:= FALSE;
			END_IF

		END_IF

	END_IF

	//Display
	//Auto Step
	IF p_tyMcParamCurr.bAutoStepEn = TRUE THEN
		fUIInRtStatOff(ADR(tyCommon.tyMain.tyBtnStep.uiRtStat));
	ELSE
		fUIInRtStatHide(ADR(tyCommon.tyMain.tyBtnStep.uiRtStat));
		fUIInRtStatHide(ADR(tyCommon.tyMain.tyBtnStep.uiMaskRtStat));
	END_IF

	//Mask
	IF (p_bAlarmErr = TRUE) OR (bUIManualMod = TRUE) OR (p_tyDI.bSafetyRlySig = FALSE) OR (tyCommon.tyMain.tyBtnHome.uiMaskRtStat.0 = FALSE) OR eCurrPage = UIP0950Simu THEN
		fUIInRtStatOff(ADR(tyCommon.tyMain.tyBtnStart.uiMaskRtStat));
		fUIInRtStatOff(ADR(tyCommon.tyMain.tyBtnStop.uiMaskRtStat));

		fUIInRtStatOff(ADR(tyP0003MMenu.tyMMenuBtn.tyBtnAuto.uiMaskRtStat));
		IF p_tyMcParamCurr.bAutoStepEn = TRUE THEN
			fUIInRtStatOff(ADR(tyCommon.tyMain.tyBtnStep.uiMaskRtStat));
		END_IF

	ELSE

		IF p_eOpsOpsStatus = OperationsStatusRun THEN

			fUIInRtStatOff(ADR(tyCommon.tyMain.tyBtnStart.uiMaskRtStat));
			fUIInRtStatHide(ADR(tyCommon.tyMain.tyBtnStop.uiMaskRtStat));
			fUIInRtStatHide(ADR(tyCommon.tyMain.tyBtnStep.uiMaskRtStat));

			fUIInRtStatOff(ADR(tyP0003MMenu.tyMMenuBtn.tyBtnAuto.uiMaskRtStat));
			fUIInRtStatHide(ADR(tyP0003MMenu.tyMMenuBtn.tyBtnStop.uiMaskRtStat));

		ELSIF p_eOpsOpsStatus = OperationsStatusCycleStopping THEN

			fUIInRtStatHide(ADR(tyCommon.tyMain.tyBtnStart.uiMaskRtStat));
			fUIInRtStatOff(ADR(tyCommon.tyMain.tyBtnStop.uiMaskRtStat));
			fUIInRtStatHide(ADR(tyCommon.tyMain.tyBtnStep.uiMaskRtStat));

			fUIInRtStatHide(ADR(tyP0003MMenu.tyMMenuBtn.tyBtnAuto.uiMaskRtStat));
			fUIInRtStatOff(ADR(tyP0003MMenu.tyMMenuBtn.tyBtnStop.uiMaskRtStat));

		ELSIF p_eOpsOpsStatus = OperationsStatusStep THEN

			fUIInRtStatHide(ADR(tyCommon.tyMain.tyBtnStart.uiMaskRtStat));
			fUIInRtStatHide(ADR(tyCommon.tyMain.tyBtnStop.uiMaskRtStat));

			IF p_eOpsStatus = Busy THEN
				fUIInRtStatOff(ADR(tyCommon.tyMain.tyBtnStep.uiMaskRtStat));
			ELSE
				fUIInRtStatHide(ADR(tyCommon.tyMain.tyBtnStep.uiMaskRtStat));
			END_IF

		ELSE

			fUIInRtStatHide(ADR(tyCommon.tyMain.tyBtnStart.uiMaskRtStat));
			fUIInRtStatOff(ADR(tyCommon.tyMain.tyBtnStop.uiMaskRtStat));

			fUIInRtStatHide(ADR(tyCommon.tyMain.tyBtnStep.uiMaskRtStat));

			fUIInRtStatHide(ADR(tyP0003MMenu.tyMMenuBtn.tyBtnAuto.uiMaskRtStat));
			fUIInRtStatOff(ADR(tyP0003MMenu.tyMMenuBtn.tyBtnStop.uiMaskRtStat));

		END_IF

	END_IF

END_ACTION
```

#### Act_OptC0005StatBarCtrl.st
```iecst
ACTION Act_OptC0005StatBarCtrl:

	//Error / Warning / Info
	IF p_bAlarmErr = TRUE OR p_bAlarmWarning = TRUE OR p_bAlarmInfo = TRUE THEN

		fbErrBlinkTm(IN := TRUE);
		IF fbErrBlinkTm.Q = TRUE THEN
			fbErrBlinkTm(IN := FALSE);

			IF p_bAlarmErr = TRUE THEN

				IF tyCommon.tyMain.tyBitmapStatBar.usiValueIdx = 1 OR tyCommon.tyMain1.tyBitmapStatBar.usiValueIdx = 1 THEN
					tyCommon.tyMain.tyBitmapStatBar.usiValueIdx		:= 0;
					tyCommon.tyMain1.tyBitmapStatBar.usiValueIdx	:= 0;
				ELSE
					tyCommon.tyMain.tyBitmapStatBar.usiValueIdx		:= 1;
					tyCommon.tyMain1.tyBitmapStatBar.usiValueIdx	:= 1;
				END_IF

			ELSE

				IF tyCommon.tyMain.tyBitmapStatBar.usiValueIdx = 3 OR tyCommon.tyMain1.tyBitmapStatBar.usiValueIdx = 3  THEN
					tyCommon.tyMain.tyBitmapStatBar.usiValueIdx		:= 0;
					tyCommon.tyMain1.tyBitmapStatBar.usiValueIdx	:= 0;
				ELSE
					tyCommon.tyMain.tyBitmapStatBar.usiValueIdx		:= 3;
					tyCommon.tyMain1.tyBitmapStatBar.usiValueIdx	:= 3;
				END_IF

			END_IF

		END_IF

	//Safety Relay Signal Activated
	ELSIF p_tyDI.bSafetyRlySig = FALSE THEN

		fbRstBlinkTm(IN := TRUE);
		IF fbRstBlinkTm.Q = TRUE THEN
			fbRstBlinkTm(IN := FALSE);

			IF tyCommon.tyMain.tyBitmapStatBar.usiValueIdx = 5 OR tyCommon.tyMain1.tyBitmapStatBar.usiValueIdx = 5 THEN
				tyCommon.tyMain.tyBitmapStatBar.usiValueIdx		:= 6;
				tyCommon.tyMain1.tyBitmapStatBar.usiValueIdx	:= 6;
			ELSE
				tyCommon.tyMain.tyBitmapStatBar.usiValueIdx		:= 5;
				tyCommon.tyMain1.tyBitmapStatBar.usiValueIdx	:= 5;
			END_IF

		END_IF

	//Manual Running
	ELSIF bUIManualMod THEN
		tyCommon.tyMain.tyBitmapStatBar.usiValueIdx		:= 0;
		tyCommon.tyMain1.tyBitmapStatBar.usiValueIdx	:= 0;

	//Operation Cycle Stopping
	ELSIF p_eOpsOpsStatus = OperationsStatusCycleStopping OR p_eSimuSimuStatus = SimulationsStatusCycleStopping THEN

		fbStopBlinkTm(IN := TRUE);
		IF fbStopBlinkTm.Q = TRUE THEN
			fbStopBlinkTm(IN := FALSE);

			IF tyCommon.tyMain.tyBitmapStatBar.usiValueIdx = 1 OR tyCommon.tyMain1.tyBitmapStatBar.usiValueIdx = 1  THEN
				tyCommon.tyMain.tyBitmapStatBar.usiValueIdx		:= 2;
				tyCommon.tyMain1.tyBitmapStatBar.usiValueIdx	:= 2;
			ELSE
				tyCommon.tyMain.tyBitmapStatBar.usiValueIdx		:= 1;
				tyCommon.tyMain1.tyBitmapStatBar.usiValueIdx	:= 1;
			END_IF

		END_IF

	//Operation Stepping
	ELSIF p_eOpsOpsStatus = OperationsStatusStep OR p_eSimuSimuStatus = SimulationsStatusRun THEN
		tyCommon.tyMain.tyBitmapStatBar.usiValueIdx		:= 3;
		tyCommon.tyMain1.tyBitmapStatBar.usiValueIdx	:= 3;

	//Operation Running
	ELSIF p_eOpsOpsStatus = OperationsStatusRun THEN
		tyCommon.tyMain.tyBitmapStatBar.usiValueIdx		:= 2;
		tyCommon.tyMain1.tyBitmapStatBar.usiValueIdx	:= 2;

	//Standby
	ELSE
		tyCommon.tyMain.tyBitmapStatBar.usiValueIdx		:= 0;
		tyCommon.tyMain1.tyBitmapStatBar.usiValueIdx	:= 0;
	END_IF

END_ACTION
```

#### Act_OptC0005ChgPage.st
```iecst
ACTION Act_OptC0005ChgPage:

	//Control Alarm and Warning
	IF tyCommon.tyMain.tyHotspotNaviStart.bRtCompl = TRUE THEN
		tyCommon.tyMain.tyHotspotNaviStart.bRtCompl := FALSE;

		IF p_bAlarmErr = TRUE OR p_bAlarmWarning THEN
			eChgPage  := UIP0600Alm;
		END_IF

	END_IF

	//Display Alarm Button Control
//	tyCommon.tyMain.tyBtnAlarm.uiRtStat.0		:= NOT (p_bAlarmErr OR p_bAlarmWarning) ;
	tyCommon.tyMain.tyHotspotNaviStart.uiRtStat.0 := tyCommon.tyMain.tyBtnStart.uiMaskRtStat.0;
	//Mask Control
//	tyCommon.tyMain.tyBtnAlarm.uiMaskRtStat.0	:= NOT ((p_bAlarmErr OR p_bAlarmWarning) AND (eCurrPage = UIP0600Alm));

END_ACTION
```

#### Act_OptC0007Notif.st
```iecst
ACTION Act_OptC0007Notif:

	//Display
	//User Level
	tyCommon.tyNotif.tyTxtUsrLv.usiValueIdx	:= UDINT_TO_USINT(p_tyUsrMgmtCurrUsr.eUsrLvl);
	tyCommon.tyNotif.tyStringUsrNm.sValue	:= p_tyUsrMgmtCurrUsr.sUsrNm;
	tyCommon.tyNotif.tyTxtLFMc.uiRtStat.0	:= NOT (p_tyNtParamCurr.bLFPrep AND p_tyMcParamCurr.bLFEn);

	IF p_tyNtParamCurr.bLFUsrSetPrep = TRUE THEN
		IF p_tyMcParamCurr.bLFLeaderMc = TRUE THEN
			tyCommon.tyNotif.tyTxtLFMc.usiValueIdx		:= 0;
		ELSE
			tyCommon.tyNotif.tyTxtLFMc.usiValueIdx		:= 1;
		END_IF
	END_IF

	//Show Info
	tyCommon.tyNotif.tyBitmapShowInfo.uiRtStat.0	:= p_bAlarmInfo = FALSE;
	tyCommon.tyNotif.tyHotspotShowInfo.uiRtStat.0	:= p_bAlarmInfo = FALSE;

	//Control
	IF tyCommon.tyNotif.tyLyr.uiRtStat.0 = FALSE THEN

		IF tyCommon.tyNotif.tyHotspotClose.bRtCompl = TRUE THEN
			tyCommon.tyNotif.tyHotspotClose.bRtCompl	:= FALSE;

			fUIInRtStatHide(ADR(tyCommon.tyNotif.tyLyr.uiRtStat));

		ELSIF tyCommon.tyNotif.tyHotspotShowInfo.bRtCompl = TRUE THEN
			tyCommon.tyNotif.tyHotspotShowInfo.bRtCompl	:= FALSE;

			fUIInRtStatOff(ADR(tyCommon.tyInfo.tyLyr.uiRtStat));
			fUIInRtStatHide(ADR(tyCommon.tyNotif.tyLyr.uiRtStat));

		END_IF

	END_IF

END_ACTION
```

#### Act_OptC0009Info.st
```iecst
ACTION Act_OptC0009Info:

	//Display
	IF EDGEPOS(p_bAlarmInfo) THEN
		fUIInRtStatOff(ADR(tyCommon.tyInfo.tyLyr.uiRtStat));
	END_IF

	IF EDGENEG(p_bAlarmInfo) THEN
		fUIInRtStatHide(ADR(tyCommon.tyInfo.tyLyr.uiRtStat));
		tyCommon.tyInfo.tyStringInfo.sValue		:= '';
		tyCommon.tyInfo.tyHotspotClose.bRtCompl	:= FALSE;
	END_IF

	IF tyCommon.tyInfo.tyHotspotClose.bRtCompl = TRUE THEN
		tyCommon.tyInfo.tyHotspotClose.bRtCompl	:= FALSE;
		fUIInRtStatHide(ADR(tyCommon.tyInfo.tyLyr.uiRtStat));

	ELSIF p_bAlarmInfo THEN
		tyCommon.tyInfo.tyStringInfo.sValue	:= p_sAlarmInfoMsg;

	END_IF

END_ACTION
```

#### Act_EntP0000Disp.st
```iecst
ACTION Act_EntP0000Disp:

	//Access Address
	p_tyP0000SSaver ACCESS ADR(tyP0000SSaver.tySSaver);

	p_tyC0008MsgBox ACCESS ADR(tyP0000SSaver.tyMsgBoxHide);
END_ACTION
```

#### Act_OptP0000McStatus.st
```iecst
ACTION Act_OptP0000McStatus:

	IF p_bAlarmErr = TRUE THEN
		tyP0000SSaver.tySSaver.tyTxtMcStat.usiValueIdx	:= 6;

	ELSIF p_bAlarmWarning = TRUE THEN
		tyP0000SSaver.tySSaver.tyTxtMcStat.usiValueIdx	:= 7;

	ELSIF p_eOpsOpsStatus = OperationsStatusRun THEN

		tyP0000SSaver.tySSaver.tyTxtMcStat.usiValueIdx	:= 1;

	ELSIF p_eSimuSimuStatus = SimulationsStatusRun THEN
		tyP0000SSaver.tySSaver.tyTxtMcStat.usiValueIdx	:= 5;

	ELSIF bUIManualMod = TRUE THEN
		tyP0000SSaver.tySSaver.tyTxtMcStat.usiValueIdx	:= 3;

	ELSE
		tyP0000SSaver.tySSaver.tyTxtMcStat.usiValueIdx	:= 2;

	END_IF

END_ACTION
```

#### Act_OptP0000RunningNm.st
```iecst
ACTION Act_OptP0000RunningNm:

	fbSSaverTm(IN := TRUE , PT := T#2s);

	IF EDGEPOS(fbSSaverTm.Q = FALSE) THEN
		CASE uiSSaverCnt OF
			0:
				tyP0000SSaver.tySSaver.tyTxtMcNm.sValue	:= CONCAT(p_tyMcParamCurr.sMcNm , '                                        ');
			1:
				tyP0000SSaver.tySSaver.tyTxtMcNm.sValue	:= CONCAT('          ' , CONCAT(p_tyMcParamCurr.sMcNm , '                              '));
			2:
				tyP0000SSaver.tySSaver.tyTxtMcNm.sValue	:= CONCAT('                    ' , CONCAT(p_tyMcParamCurr.sMcNm , '                    '));
			3:
				tyP0000SSaver.tySSaver.tyTxtMcNm.sValue	:= CONCAT('                              ' , CONCAT(p_tyMcParamCurr.sMcNm , '          '));
			4:
				tyP0000SSaver.tySSaver.tyTxtMcNm.sValue	:= CONCAT('                                        ' , p_tyMcParamCurr.sMcNm);
			5:
				tyP0000SSaver.tySSaver.tyTxtMcNm.sValue	:= CONCAT('                              ' , CONCAT(p_tyMcParamCurr.sMcNm , '          '));
			6:
				tyP0000SSaver.tySSaver.tyTxtMcNm.sValue	:= CONCAT('                    ' , CONCAT(p_tyMcParamCurr.sMcNm , '                    '));
			7:
				tyP0000SSaver.tySSaver.tyTxtMcNm.sValue	:= CONCAT('          ' , CONCAT(p_tyMcParamCurr.sMcNm , '                              '));

		END_CASE

	END_IF

	IF fbSSaverTm.Q = TRUE THEN
		fbSSaverTm(IN := FALSE);
		uiSSaverCnt	:= uiSSaverCnt + 1;
		IF uiSSaverCnt = 8 THEN
			uiSSaverCnt	:= 0;
		END_IF
	END_IF

END_ACTION
```

#### Act_OptP0000DisableSSaver.st
```iecst
ACTION Act_OptP0000DisableSSaver:

	IF p_tyNtParamCurr.bSSaverPrep = FALSE OR p_tyMcParamCurr.bSSaverEn = FALSE THEN

		IF tyProperty.tyVisu.uiScreenSaverRemainTm < 5 THEN
			tyProperty.tyVisu.uiSSaverTm	:= 9;
		ELSE
			tyProperty.tyVisu.uiSSaverTm	:= 10;
		END_IF

	END_IF

	IF EDGEPOS(p_tyNtParamCurr.bSSaverPrep AND p_tyMcParamCurr.bSSaverEn) THEN
		tyProperty.tyVisu.uiSSaverTm	:= p_tyMcParamCurr.uiSSaverTmInSec;
	END_IF

END_ACTION
```

#### Act_OptP0000StatDisp.st
```iecst
ACTION Act_OptP0000StatDisp:

	//Error / Warning / Info
	IF p_bAlarmErr = TRUE OR p_bAlarmWarning = TRUE OR p_bAlarmInfo = TRUE THEN

		fbErrBlinkTm(IN := TRUE);
		IF fbErrBlinkTm.Q = TRUE THEN
			fbErrBlinkTm(IN := FALSE);

			IF p_bAlarmErr THEN

				IF tyP0000SSaver.tySSaver.tyBitmapStat.usiValueIdx = 1 THEN
					tyP0000SSaver.tySSaver.tyBitmapStat.usiValueIdx	:= 0;
				ELSE
					tyP0000SSaver.tySSaver.tyBitmapStat.usiValueIdx	:= 1;
				END_IF

			ELSE

				IF tyP0000SSaver.tySSaver.tyBitmapStat.usiValueIdx = 3 THEN
					tyP0000SSaver.tySSaver.tyBitmapStat.usiValueIdx	:= 0;
				ELSE
					tyP0000SSaver.tySSaver.tyBitmapStat.usiValueIdx	:= 3;
				END_IF

			END_IF

		END_IF

	//Safety Relay Signal Activated
	ELSIF p_tyDI.bSafetyRlySig = FALSE THEN

		fbRstBlinkTm(IN := TRUE);
		IF fbRstBlinkTm.Q = TRUE THEN
			fbRstBlinkTm(IN := FALSE);

			IF tyP0000SSaver.tySSaver.tyBitmapStat.usiValueIdx = 5 THEN
				tyP0000SSaver.tySSaver.tyBitmapStat.usiValueIdx	:= 6;
			ELSE
				tyP0000SSaver.tySSaver.tyBitmapStat.usiValueIdx	:= 5;
			END_IF

		END_IF

	//Manual Running
	ELSIF bUIManualMod THEN
		tyP0000SSaver.tySSaver.tyBitmapStat.usiValueIdx	:= 7;

	//Operation Cycle Stopping
	ELSIF p_eOpsOpsStatus = OperationsStatusCycleStopping OR p_eSimuSimuStatus = SimulationsStatusCycleStopping THEN

		fbStopBlinkTm(IN := TRUE);
		IF fbStopBlinkTm.Q = TRUE THEN
			fbStopBlinkTm(IN := FALSE);

			IF tyP0000SSaver.tySSaver.tyBitmapStat.usiValueIdx = 1 THEN
				tyP0000SSaver.tySSaver.tyBitmapStat.usiValueIdx	:= 2;
			ELSE
				tyP0000SSaver.tySSaver.tyBitmapStat.usiValueIdx	:= 1;
			END_IF

		END_IF

	//Operation Stepping
	ELSIF p_eOpsOpsStatus = OperationsStatusStep THEN
		tyP0000SSaver.tySSaver.tyBitmapStat.usiValueIdx	:= 3;

	//Operation Running
	ELSIF p_eOpsOpsStatus = OperationsStatusRun OR p_eSimuSimuStatus = SimulationsStatusRun THEN
		tyP0000SSaver.tySSaver.tyBitmapStat.usiValueIdx	:= 2;

	//Standby
	ELSE
		tyP0000SSaver.tySSaver.tyBitmapStat.usiValueIdx	:= 0;

	END_IF

END_ACTION
```

#### Act_OptP0000TouchTimer.st
```iecst
ACTION Act_OptP0000TouchTimer:

	IF bLoginSuccess AND p_tyNtParamCurr.bAutoLogoutPrep AND p_tyMcParamCurr.bAutoLogoutEn THEN

		fbTouchTm();

		fbAutoLogoutTm(IN:= NOT fbTouchTm.bPressed, PT:=DINT_TO_TIME(p_tyMcParamCurr.diAutoLogoutTmInSec));

		//Reset Time When Pressed
		IF fbTouchTm.bPressed THEN
			fbAutoLogoutTm(IN:=FALSE);
		END_IF

		//Auto Logout
		IF fbAutoLogoutTm.Q THEN

			bPromptSessionExp	:= TRUE;
			p_tyC0008MsgBox ACCESS ADR(tyP0000SSaver.tyMsgBoxLoginAsk);

			IF bChgPageDone=FALSE THEN

				IF eCurrPage<>UIP0003MMenu THEN // Previous - UIP0002Menu
					CASE eCurrPage OF

						UIP0900GenIn, UIP0910GenOut, UIP0920MtrNPneuCtrl,UIP0921Shutter, UIP0922Stopper, UIP0933PusherConv, UIP0934AW, UIP0935Lifter, UIP0936Trav, UIP0940CommCtrl, UIP0950Simu:

							eChgPage	:=	UIP0003MMenu; // Previous - UIP0002Menu

							tyP0002Menu.tyMenu.tyBtnMnlRst.bRtCompl := TRUE ;

							bChgPageDone	:= TRUE;

						UIP1000Lang, UIP1021McSetGen, UIP1022McSetVComm, UIP1023McSetHComm, UIP1024McSetAntiGap, UIP1026McSetTeach,UIP1030MagSet, UIP1031MagSetTeach,UIP1040ProdSet, UIP1050LFSet:

							IF tyCommon.tySet.tyBtnSave.uiMaskRtStat.0 = FALSE THEN

								eChgPage	:= UIP0003MMenu; // Previous - UIP0002Menu

								bChgPageDone	:= TRUE;

							ELSE

								eChgPage	:= UIP0003MMenu; //	:= UIP0002Menu;

								IF eCurrPage= UIP1021McSetGen THEN

									tyP1021McSetGen.tyMsgBoxExitAsk.tyBtnYes.bRtCompl := TRUE;

									bChgPageDone	:= TRUE;

								ELSIF eCurrPage= UIP1022McSetVComm THEN

									tyP1022McSetVComm.tyMsgBoxExitAsk.tyBtnYes.bRtCompl := TRUE;

									bChgPageDone	:= TRUE;

								ELSIF eCurrPage= UIP1023McSetHComm THEN

									tyP1023McSetHComm.tyMsgBoxExitAsk.tyBtnYes.bRtCompl := TRUE;

									bChgPageDone	:= TRUE;

								ELSIF eCurrPage= UIP1024McSetAntiGap THEN

									tyP1024McSetAntiGap.tyMsgBoxExitAsk.tyBtnYes.bRtCompl := TRUE;

									bChgPageDone	:= TRUE;

								ELSIF eCurrPage= UIP1026McSetTeach THEN

									tyP1026McSetTeach.tyMsgBoxExitAsk.tyBtnYes.bRtCompl := TRUE;

									bChgPageDone	:= TRUE;

								ELSIF eCurrPage= UIP1030MagSet THEN

									tyP1030MagSet.tyMsgBoxExitAsk.tyBtnYes.bRtCompl := TRUE;

									bChgPageDone	:= TRUE;

								ELSIF eCurrPage= UIP1031MagSetTeach THEN

									tyP1031MagSetTeach.tyMsgBoxExitAsk.tyBtnYes.bRtCompl := TRUE;

									bChgPageDone	:= TRUE;

								ELSE  //language page
									bChgPageDone	:= TRUE;
								END_IF

							END_IF

						ELSE
							eChgPage		:= UIP0003MMenu; ;//eChgPage		:= UIP0002Menu;

							bChgPageDone	:= TRUE;

					END_CASE

				ELSE
					bChgPageDone	:= TRUE;
				END_IF

			END_IF

			IF bChgPageDone THEN

				eUsrMgmtAct	:= UsrMgmtActLogout;

				IF p_eUsrMgmtStat = UsrMgmtActLogout AND p_eUsrMgmtStatus = Done THEN
					eUsrMgmtAct	:= UsrMgmtActIdle;

					bLoginSuccess	:= FALSE;

					bChgPageDone	:= FALSE;

					fbAutoLogoutTm(IN:=FALSE);

				END_IF

			END_IF

		END_IF

	ELSE
		fbAutoLogoutTm(IN:=FALSE);
		bChgPageDone	:= FALSE;
	END_IF

	//Prompt Relogin After Auto Logout
	IF tyP0000SSaver.tyMsgBoxLoginAsk.tyBtnYes.bRtCompl = TRUE THEN
		tyP0000SSaver.tyMsgBoxLoginAsk.tyBtnYes.bRtCompl 	:= FALSE;
		tyP0000SSaver.tyMsgBoxLoginAsk.tyBtnYes.bValue		:= FALSE;
		p_tyC0008MsgBox ACCESS ADR(tyP0000SSaver.tyMsgBoxHide);
		bPromptSessionExp :=FALSE;

	ELSIF tyP0000SSaver.tyMsgBoxLoginAsk.tyBtnNo.bRtCompl = TRUE THEN
		tyP0000SSaver.tyMsgBoxLoginAsk.tyBtnNo.bRtCompl 	:= FALSE;
		tyP0000SSaver.tyMsgBoxLoginAsk.tyBtnNo.bValue		:= FALSE;
		p_tyC0008MsgBox ACCESS ADR(tyP0000SSaver.tyMsgBoxHide);
		eChgPage		:= UIP0100Login;
		bPromptSessionExp :=FALSE;
	END_IF

END_ACTION
```

#### Act_OptP0000Hermes.st
```iecst
ACTION Act_OptP0000Hermes: //Can receive at anytime, at any Page

	//SendBordInfo can be received at anytime, at any Page
	IF (p_bRcvBoardInfoIncompl AND tyCommon.tyInfo.tyHotspotClose.bRtCompl = TRUE) OR EDGENEG (p_bRcvBoardInfoOk) OR tyP0201OpsTravLifter.tyOps.tyBtnQueryBoardInfo.bValue = FALSE THEN //Reset
		bQueryBoardInfo := FALSE;
		tyP0201OpsTravLifter.tyOps.tyBtnQueryBoardInfo.bValue := FALSE;
	END_IF

	//Reset QueryWorkOrderInfo when Close C0009 Info
	IF EDGEPOS (tyCommon.tyInfo.tyHotspotClose.bRtCompl = TRUE OR tyP0201OpsTravLifter.tyOps.tyBtnQueryWorkOrderInfo.bValue = FALSE OR p_bRcvWorkOrderInfo1) THEN
		bQueryWorkOrderInfo := FALSE;
		tyP0201OpsTravLifter.tyOps.tyBtnQueryWorkOrderInfo.bValue := FALSE;
	END_IF

	//Configure update can happen at anytime, at any Page (Can modify to Reset this when User Press tyCommon.tyInfo.tyHotspotClose.bRtCompl)
	IF p_bRmtUpdateUIData = TRUE OR p_bSvyUpdateUIData = TRUE THEN

		//Update UI Upstream Configure
		tyP1023McSetHComm.tyUSHermesA.tyNumSndAliveTm.diValue		:= TIME_TO_DINT(p_tyHermesConfiguration.a_tyUSParam[0].tSndAlive);
		tyP1023McSetHComm.tyUSHermesA.tyNumLaneID.diValue			:= INT_TO_DINT(p_tyHermesConfiguration.a_tyUSParam[0].iLaneID);
		tyP1023McSetHComm.tyUSHermesA.tyNumHostPort.diValue			:= UINT_TO_DINT(p_tyHermesConfiguration.a_tyUSParam[0].uiHostPort);
		tyP1023McSetHComm.tyUSHermesA.tyStringHostAddr.sValue		:= p_tyHermesConfiguration.a_tyUSParam[0].sHostAddress;
		tyP1023McSetHComm.tyUSHermesA.tyBtnCheckAliveResponse.bValue	:= p_tyHermesConfiguration.a_tyUSParam[0].bFeatureCheckAliveResponse;
		tyP1023McSetHComm.tyUSHermesA.tyBtnCmpTypeId.bValue			:= p_tyHermesConfiguration.a_tyUSParam[0].bCmpTypeId;
		tyP1023McSetHComm.tyUSHermesA.tyBtnCmpParam.bValue			:= p_tyHermesConfiguration.a_tyUSParam[0].bCmpParam;
		tyP1023McSetHComm.tyUSHermesA.tyBtnOverWrite.bValue			:= p_tyHermesConfiguration.a_tyUSParam[0].bOverwrite;
		tyP1023McSetHComm.tyUSHermesA.tyBtnBoardForecast.bValue		:= p_tyHermesConfiguration.a_tyUSParam[0].bFeatureBoardForecast;//new
		tyP1023McSetHComm.tyUSHermesA.tyBtnQueryBoardInfo.bValue		:= p_tyHermesConfiguration.a_tyUSParam[0].bFeatureQueryBoardInfo;//new

		tyP1023McSetHComm.tyUSHermesB.tyNumSndAliveTm.diValue		:= TIME_TO_DINT(p_tyHermesConfiguration.a_tyUSParam[1].tSndAlive);
		tyP1023McSetHComm.tyUSHermesB.tyNumLaneID.diValue			:= INT_TO_DINT(p_tyHermesConfiguration.a_tyUSParam[1].iLaneID);
		tyP1023McSetHComm.tyUSHermesB.tyNumHostPort.diValue			:= UINT_TO_DINT(p_tyHermesConfiguration.a_tyUSParam[1].uiHostPort);
		tyP1023McSetHComm.tyUSHermesB.tyStringHostAddr.sValue		:= p_tyHermesConfiguration.a_tyUSParam[1].sHostAddress;
		tyP1023McSetHComm.tyUSHermesB.tyBtnCheckAliveResponse.bValue	:= p_tyHermesConfiguration.a_tyUSParam[1].bFeatureCheckAliveResponse;
		tyP1023McSetHComm.tyUSHermesB.tyBtnCmpTypeId.bValue			:= p_tyHermesConfiguration.a_tyUSParam[1].bCmpTypeId;
		tyP1023McSetHComm.tyUSHermesB.tyBtnCmpParam.bValue			:= p_tyHermesConfiguration.a_tyUSParam[1].bCmpParam;
		tyP1023McSetHComm.tyUSHermesB.tyBtnOverWrite.bValue			:= p_tyHermesConfiguration.a_tyUSParam[1].bOverwrite;
		tyP1023McSetHComm.tyUSHermesB.tyBtnBoardForecast.bValue		:= p_tyHermesConfiguration.a_tyUSParam[1].bFeatureBoardForecast;//new
		tyP1023McSetHComm.tyUSHermesB.tyBtnQueryBoardInfo.bValue		:= p_tyHermesConfiguration.a_tyUSParam[1].bFeatureQueryBoardInfo;//new

		//Update UI Supervisory Configure
		tyP1022McSetVComm.tyVComSvy.tyNumSndAliveTm.diValue	    	:= TIME_TO_DINT(p_tyHermesConfiguration.tySvyParam.tSndAlive);
		tyP1022McSetVComm.tyVComSvy.tyNumSvySystemPort.diValue	    := UINT_TO_DINT(p_tyHermesConfiguration.tySvyParam.uiSvySvstemPort);
		tyP1022McSetVComm.tyVComSvy.tyBtnConfiguration.bValue		:= p_tyHermesConfiguration.tySvyParam.bFeatureConfiguration;
		tyP1022McSetVComm.tyVComSvy.tyBtnCheckAliveResponse.bValue	:= p_tyHermesConfiguration.tySvyParam.bFeatureCheckAliveResponse;
		tyP1022McSetVComm.tyVComSvy.tyBtnBoardTracking.bValue		:= p_tyHermesConfiguration.tySvyParam.bFeatureBoardTracking;
		tyP1022McSetVComm.tyVComSvy.tyBtnQueryWorkOrderInfo.bValue	:= p_tyHermesConfiguration.tySvyParam.bFeatureQueryWorkOrderInfo;
		tyP1022McSetVComm.tyVComSvy.tyBtnSendWorkOrderInfo.bValue   := p_tyHermesConfiguration.tySvyParam.bFeatureSendWorkOrderInfo;

		//Update UI Mc Name and Backup Mc Name of P1021
		tyP1021McSetGen.tyGen.tyStringMcNm.sValue			    	:= p_tyMcParamCurr.sMcNm; //String[30] doesnt tally with MachineId String[80] currently.
		tyP1021McSetGen.tyGenBkUp.tyStringMcNm	                    := tyP1021McSetGen.tyGen.tyStringMcNm;

		//Update Backup Param P1022
		tyP1022McSetVComm.tyVComSelBkUp	    := tyP1022McSetVComm.tyVComSel;
		tyP1022McSetVComm.tyVComSvyBkUp	    := tyP1022McSetVComm.tyVComSvy;
		tyP1022McSetVComm.tyLFBkUp		    := tyP1022McSetVComm.tyLF;

		//Update Backup Param P1023
		tyP1023McSetHComm.tyUSSelABkUp		:= tyP1023McSetHComm.tyUSSelA;
		tyP1023McSetHComm.tyUSSMEMAABkUp	:= tyP1023McSetHComm.tyUSSMEMAA;
		tyP1023McSetHComm.tyUSHermesABkUp	:= tyP1023McSetHComm.tyUSHermesA;

		tyP1023McSetHComm.tyUSSelBBkUp		:= tyP1023McSetHComm.tyUSSelB;
		tyP1023McSetHComm.tyUSSMEMABBkUp	:= tyP1023McSetHComm.tyUSSMEMAB;
		tyP1023McSetHComm.tyUSHermesBBkUp	:= tyP1023McSetHComm.tyUSHermesB;

	END_IF

END_ACTION
```

#### Act_EntP0001Disp.st
```iecst
ACTION Act_EntP0001Disp:

	//UI Property Access
	p_tyVisu ACCESS ADR(tyProperty.tyVisu);

	p_tyKeypad ACCESS ADR(tyProperty.tyKeypad);

	p_tyTxtSnippets ACCESS ADR(tyProperty.tyUITxtSnippets);

	p_tyC0008MsgBox ACCESS ADR(tyP0001Startup.tyMsgBoxHide);

	//Access Address
	p_tyP0001Startup ACCESS ADR(tyP0001Startup.tyStartup);

	p_tyP0001Initial ACCESS ADR(tyP0001Startup.tyInitial);

	fUIInRtStatHide(ADR(tyP0001Startup.tyInitial.tyLyr.uiRtStat));

END_ACTION
```

#### Act_OptP0001Startup.st
```iecst
ACTION Act_OptP0001Startup:
	//Gloabal IP assign
	g_sIPAddress.sSetIPAddress			:= sSetIPAddr;
	g_sIPAddress.sSetSubnetMask			:= sSetSubnetMask;
	g_sIPAddress.sSelectedNetworkMode	:= sSelectedNetworkMode;
	g_sIPAddress.sTempIpAddress			:= sTempIPAddr;
	g_sIPAddress.sTempSubnetMask		:= sTempSubnetMask;
	g_sIPAddress.sTempNetworkMode		:= sTempNetworkMode;

	//Temp Network Mode
	IF udiTempEthMode = 0 THEN
		sTempNetworkMode := 'Manually Set IP';
	ELSIF udiTempEthMode = 1 THEN
		sTempNetworkMode := 'Get IP from DHCP Server';
	END_IF
	//Current Network Mode
	IF usiNetworkModeSelected = 0 THEN
		sSelectedNetworkMode	:= 'Manually Set IP';
	ELSIF usiNetworkModeSelected = 1 THEN
		sSelectedNetworkMode	:= 'Get IP from DHCP Server';
	END_IF
	//Screen Saver
	p_tyP0000SSaver ACCESS ADR(tyP0000SSaver.tySSaver);

	IF (eChgPage = UIP0001Startup) AND (eCurrPage = UIP0001Startup) THEN

		eStartupAct		:= StartupActRun;

		IF p_eStartupStat = StartupActRun AND p_eStartupStatus = Done THEN
			eStartupAct	:= StartupActIdle;

			IF p_bAlarmErr OR p_bAlarmWarning THEN
				eChgPage	:= UIP0600Alm;
			ELSE
				eChgPage	:= UIP0003MMenu; // UIP0002Menu;
			END_IF

		END_IF

	END_IF

	tyP0001Startup.tyStartup.tyBarGraphStartup.iValue	:= DINT_TO_INT(p_eStartupStep + 1);
	tyP0001Startup.tyStartup.tyTxtStartupStat.sTxt		:= p_sStartupStepTxt;

	//IP Config
	IF DiagCpuIsSimulated() = FALSE THEN
	IF p_eStartupStep>1 THEN

		IF p_bStartupGetConfigDone THEN
			IF bTempAddrFillDone=FALSE THEN

				tyMcParamWr:= p_tyMcParamCurr;

				sTempIPAddr 	:= p_sHWInfoIPAddr;
				sTempSubnetMask	:= p_sHWInfoSubnetMask;
				udiTempEthMode	:= p_udiHWInfoEthMode;

				bTempAddrFillDone	:= TRUE;
			END_IF
		END_IF

		IF bTempAddrFillDone THEN

			IF bIPConfigChgDone=FALSE THEN

				IF  (p_tyMcParamCurr.eNetworkMod = UDINT_TO_DINT(udiTempEthMode)) AND (p_tyMcParamCurr.sIPAddr = sTempIPAddr) AND (p_tyMcParamCurr.sSubnetMask = sTempSubnetMask) THEN

					p_tyC0008MsgBox ACCESS ADR(tyP0001Startup.tyMsgBoxHide);
				ELSE
					IF p_bStartupMismatchSetConfigDone THEN

						IF (p_tyMcParamCurr.eNetworkMod <> UDINT_TO_DINT(udiTempEthMode)) THEN
							tyP0001Startup.tyMsgBoxIPConfig.tyTxtMsg.usiValueIdx := 189;// 114;
						ELSIF (p_tyMcParamCurr.sIPAddr <> sTempIPAddr) AND (p_tyMcParamCurr.sSubnetMask <> sTempSubnetMask) THEN
							tyP0001Startup.tyMsgBoxIPConfig.tyTxtMsg.usiValueIdx := 186; //113;
						ELSIF (p_tyMcParamCurr.sIPAddr <> sTempIPAddr) THEN
							tyP0001Startup.tyMsgBoxIPConfig.tyTxtMsg.usiValueIdx := 187; //111;
						ELSE
							tyP0001Startup.tyMsgBoxIPConfig.tyTxtMsg.usiValueIdx := 188; //112;
						END_IF

							p_tyC0008MsgBox ACCESS ADR(tyP0001Startup.tyMsgBoxIPConfig);

					ELSE
						sSetIPAddr				:= p_tyMcParamCurr.sIPAddr;
						sSetSubnetMask			:= p_tyMcParamCurr.sSubnetMask;
						usiNetworkModeSelected	:= DINT_TO_USINT(p_tyMcParamCurr.eNetworkMod);

							bMismatchOverWriteConfig			:= TRUE;
						END_IF

					END_IF

				END_IF
			END_IF
		END_IF
	END_IF

	IF tyP0001Startup.tyMsgBoxIPConfig.tyBtnYes.bRtCompl = TRUE THEN
		tyP0001Startup.tyMsgBoxIPConfig.tyBtnYes.bRtCompl	:= FALSE;
		tyP0001Startup.tyMsgBoxIPConfig.tyBtnYes.bValue	:= FALSE;

		bIPConfigChgDone	:= TRUE;

		p_tyC0008MsgBox ACCESS ADR(tyP0001Startup.tyMsgBoxHide);

	ELSIF tyP0001Startup.tyMsgBoxIPConfig.tyBtnNo.bRtCompl = TRUE THEN

		IF (p_tyMcParamCurr.eNetworkMod <> UDINT_TO_DINT(udiTempEthMode))  THEN

			IF udiTempEthMode = DINT_TO_UDINT(IPFromDHCPServer) THEN

				bOverwriteEthMode	:= TRUE;
				bOverwriteIP 		:= FALSE;
				bOverwriteSubnet	:= FALSE;

				usiNetworkModeSelected	:= UDINT_TO_USINT(udiTempEthMode);

				tyMcParamWr.eNetworkMod	:= UDINT_TO_DINT(udiTempEthMode);

				bIPConfigChgDone	:= TRUE;

				tyP0001Startup.tyMsgBoxIPConfig.tyBtnNo.bRtCompl:= FALSE;
				tyP0001Startup.tyMsgBoxIPConfig.tyBtnNo.bValue	:= FALSE;

				p_tyC0008MsgBox ACCESS ADR(tyP0001Startup.tyMsgBoxHide);
			ELSE
				bOverwriteEthMode	:= TRUE;
				bOverwriteIP 		:= TRUE;
				bOverwriteSubnet	:= TRUE;

				usiNetworkModeSelected	:= UDINT_TO_USINT(udiTempEthMode);
				sSetIPAddr				:= sTempIPAddr;
				sSetSubnetMask			:= sTempSubnetMask;

				tyMcParamWr.eNetworkMod			:= UDINT_TO_DINT(udiTempEthMode);
				tyMcParamWr.sIPAddr				:= sTempIPAddr;
				tyMcParamWr.sSubnetMask			:= sTempSubnetMask;

				bIPConfigChgDone	:= TRUE;

				tyP0001Startup.tyMsgBoxIPConfig.tyBtnNo.bRtCompl:= FALSE;
				tyP0001Startup.tyMsgBoxIPConfig.tyBtnNo.bValue	:= FALSE;

				p_tyC0008MsgBox ACCESS ADR(tyP0001Startup.tyMsgBoxHide);
			END_IF

		ELSE

			IF (p_tyMcParamCurr.sIPAddr <> sTempIPAddr) AND (p_tyMcParamCurr.sSubnetMask <> sTempSubnetMask) THEN

				bOverwriteEthMode	:= FALSE;
				bOverwriteIP 		:= TRUE;
				bOverwriteSubnet	:= TRUE;

				sSetIPAddr		:= sTempIPAddr;
				sSetSubnetMask	:= sTempSubnetMask;

				tyMcParamWr.sIPAddr				:= sTempIPAddr;
				tyMcParamWr.sSubnetMask			:= sTempSubnetMask;

				bIPConfigChgDone	:= TRUE;

				tyP0001Startup.tyMsgBoxIPConfig.tyBtnNo.bRtCompl	:= FALSE;
				tyP0001Startup.tyMsgBoxIPConfig.tyBtnNo.bValue	:= FALSE;

				p_tyC0008MsgBox ACCESS ADR(tyP0001Startup.tyMsgBoxHide);

			ELSIF (p_tyMcParamCurr.sIPAddr <> sTempIPAddr) THEN

				bOverwriteEthMode	:= FALSE;
				bOverwriteIP 		:= TRUE;
				bOverwriteSubnet	:= FALSE;

				sSetIPAddr			:= sTempIPAddr;

				tyMcParamWr.sIPAddr	:= sTempIPAddr;

				bIPConfigChgDone	:= TRUE;

				tyP0001Startup.tyMsgBoxIPConfig.tyBtnNo.bRtCompl	:= FALSE;
				tyP0001Startup.tyMsgBoxIPConfig.tyBtnNo.bValue	:= FALSE;

				p_tyC0008MsgBox ACCESS ADR(tyP0001Startup.tyMsgBoxHide);
			ELSE

				bOverwriteEthMode	:= FALSE;
				bOverwriteIP 		:= FALSE;
				bOverwriteSubnet	:= TRUE;

				sSetSubnetMask	:= sTempSubnetMask;

				tyMcParamWr.sSubnetMask			:= sTempSubnetMask;

				bIPConfigChgDone				:= TRUE;

				tyP0001Startup.tyMsgBoxIPConfig.tyBtnNo.bRtCompl	:= FALSE;
				tyP0001Startup.tyMsgBoxIPConfig.tyBtnNo.bValue		:= FALSE;

				p_tyC0008MsgBox ACCESS ADR(tyP0001Startup.tyMsgBoxHide);
			END_IF
		END_IF
	END_IF

END_ACTION
```

#### Act_EntP0002Disp.st
```iecst
ACTION Act_EntP0002Disp:

	//Access
	p_tyC0005Main ACCESS ADR(tyCommon.tyMain);

	p_tyC0007Notif ACCESS ADR(tyCommon.tyNotif);

//	p_tyC0008MsgBox ACCESS ADR(tyP0002Menu.tyMsgBoxHide);
	IF NOT bPromptSessionExp THEN
		p_tyC0008MsgBox ACCESS ADR(tyP0002Menu.tyMsgBoxHide);
	END_IF

	p_tyC0009Info ACCESS ADR(tyCommon.tyInfo);

	p_tyP0002Menu ACCESS ADR(tyP0002Menu.tyMenu);

	//Display
	//Leader Follower
	IF p_tyNtParamCurr.bProjLaneBPrep THEN
		IF p_tyNtParamCurr.bLFPrep = TRUE AND p_tyMcParamCurr.bLFEn = TRUE AND ((NOT p_tyNtParamCurr.bLFUsrSetPrep AND p_tyNtParamCurr.bLeaderMc) OR (p_tyNtParamCurr.bLFUsrSetPrep AND p_tyMcParamCurr.bLFLeaderMc)) AND p_tyMcParamCurr.eUSCommA <> McSetCommModHermes AND p_tyMcParamCurr.eUSCommB <> McSetCommModHermes THEN
			fUIInRtStatOff(ADR(tyP0002Menu.tyMenu.tyBtnLFSet.uiRtStat));
			fUIInRtStatOff(ADR(tyP0002Menu.tyMenu.tyBtnLFCtrl.uiRtStat));
		ELSE
			fUIInRtStatHide(ADR(tyP0002Menu.tyMenu.tyBtnLFSet.uiRtStat));
			fUIInRtStatHide(ADR(tyP0002Menu.tyMenu.tyBtnLFCtrl.uiRtStat));
		END_IF
	ELSE
		IF p_tyNtParamCurr.bLFPrep = TRUE AND p_tyMcParamCurr.bLFEn = TRUE AND ((NOT p_tyNtParamCurr.bLFUsrSetPrep AND p_tyNtParamCurr.bLeaderMc) OR (p_tyNtParamCurr.bLFUsrSetPrep AND p_tyMcParamCurr.bLFLeaderMc)) AND p_tyMcParamCurr.eUSCommA <> McSetCommModHermes THEN
			fUIInRtStatOff(ADR(tyP0002Menu.tyMenu.tyBtnLFSet.uiRtStat));
			fUIInRtStatOff(ADR(tyP0002Menu.tyMenu.tyBtnLFCtrl.uiRtStat));
		ELSE
			fUIInRtStatHide(ADR(tyP0002Menu.tyMenu.tyBtnLFSet.uiRtStat));
			fUIInRtStatHide(ADR(tyP0002Menu.tyMenu.tyBtnLFCtrl.uiRtStat));
		END_IF
	END_IF

	//Login Logout Display
	IF bLoginSuccess = FALSE THEN
		tyP0002Menu.tyMenu.tyBtnLogin.usiBitmapIdx	:= 0;
		tyP0002Menu.tyMenu.tyBtnLogin.usiTxtIdx		:= 0;
	ELSE
		tyP0002Menu.tyMenu.tyBtnLogin.usiBitmapIdx	:= 1;
		tyP0002Menu.tyMenu.tyBtnLogin.usiTxtIdx		:= 1;
	END_IF

	//Oven Info
	tyP0002Menu.tyMenu.tyBtnOvenInfo.uiRtStat.0	:= NOT(p_tyNtParamCurr.bOvenInfoPrep AND p_tyMcParamCurr.bOvenEn);

	//Mask
	Act_OptP0002Mask;

//	IF p_tyMcParamCurr.bAGVComEn = FALSE THEN
//		fUIInRtStatHide(ADR(tyP0002Menu.tyMenu.tyBtnSimu.uiRtStat));
//	ELSE
//		fUIInRtStatOff(ADR(tyP0002Menu.tyMenu.tyBtnSimu.uiRtStat));
//	END_IF

END_ACTION
```

#### Act_OptP0002Mask.st
```iecst
ACTION Act_OptP0002Mask:

	tyP0002Menu.tyMenu.tyBtnOpt.uiMaskRtStat.0 					:= p_tyUsrMgmtCurrAccessRgt.bOpt;
	tyP0002Menu.tyMenu.tyBtnMcInfo.uiMaskRtStat.0 				:= p_tyUsrMgmtCurrAccessRgt.bMcInfo;
	tyP0002Menu.tyMenu.tyBtnMagInfo.uiMaskRtStat.0				:= p_tyUsrMgmtCurrAccessRgt.bMagInfo;
	tyP0002Menu.tyMenu.tyBtnOvenInfo.uiMaskRtStat.0				:= p_tyUsrMgmtCurrAccessRgt.bOvenInfo;
	tyP0002Menu.tyMenu.tyBtnAlm.uiMaskRtStat.0 					:= p_tyUsrMgmtCurrAccessRgt.bAlm;
	tyP0002Menu.tyMenu.tyBtnLogin.uiMaskRtStat.0				:= p_bOpsStatusStop;
	tyP0002Menu.tyMenu.tyBtnLFCtrl.uiMaskRtStat.0 				:= p_tyUsrMgmtCurrAccessRgt.bLFCtrl;
	tyP0002Menu.tyMenu.tyBtnGenInput.uiMaskRtStat.0				:= p_tyUsrMgmtCurrAccessRgt.bManual AND p_bOpsStatusStop;
	tyP0002Menu.tyMenu.tyBtnGenOutput.uiMaskRtStat.0			:= p_tyUsrMgmtCurrAccessRgt.bManual AND p_bOpsStatusStop;
	tyP0002Menu.tyMenu.tyBtnMovCtrl.uiMaskRtStat.0 				:= p_tyUsrMgmtCurrAccessRgt.bManual AND p_bOpsStatusStop;
	tyP0002Menu.tyMenu.tyBtnCommCtrl.uiMaskRtStat.0 			:= p_tyUsrMgmtCurrAccessRgt.bManual AND p_bOpsStatusStop;
	tyP0002Menu.tyMenu.tyBtnSimu.uiMaskRtStat.0 				:= p_tyUsrMgmtCurrAccessRgt.bSimulation AND p_bOpsStatusStop;
	tyP0002Menu.tyMenu.tyBtnProdSet.uiMaskRtStat.0 				:= p_tyUsrMgmtCurrAccessRgt.bProdSet AND p_bOpsStatusStop;
	tyP0002Menu.tyMenu.tyBtnMagSet.uiMaskRtStat.0				:= p_tyUsrMgmtCurrAccessRgt.bMagSet AND p_bOpsStatusStop;
	tyP0002Menu.tyMenu.tyBtnMcSet.uiMaskRtStat.0 				:= p_tyUsrMgmtCurrAccessRgt.bMcSet AND p_bOpsStatusStop;
	tyP0002Menu.tyMenu.tyBtnLang.uiMaskRtStat.0 				:= p_tyUsrMgmtCurrAccessRgt.bLang AND p_bOpsStatusStop;
	tyP0002Menu.tyMenu.tyBtnUsrMgmt.uiMaskRtStat.0 				:= p_tyUsrMgmtCurrAccessRgt.bUsrMgmt AND p_bOpsStatusStop;
	tyP0002Menu.tyMenu.tyBtnLFSet.uiMaskRtStat.0 				:= p_tyUsrMgmtCurrAccessRgt.bLFSet AND p_bOpsStatusStop;

	tyP0002Menu.tyMenu.tyBitmapMaskProdSetLCS.uiMaskRtStat.0	:= NOT(p_tyNtParamCurr.bLCSManageRcpPrep AND p_tyMcParamCurr.bLCSManageRcpEn);

//	IF p_tyNtParamCurr.eProjMag = ULMagTriple THEN
//		tyP0002Menu.tyMenu.tyBtnProdSel.uiMaskRtStat.0 	:= p_tyUsrMgmtCurrAccessRgt.bProdSel AND p_bOpsStatusStop AND NOT(p_bBuffer1MagPresent OR p_bBuffer2MagPresent OR p_bBuffer3MagPresent);
//		tyP0002Menu.tyMenu.tyBtnMagSel.uiMaskRtStat.0	:= p_tyUsrMgmtCurrAccessRgt.bMagSel AND p_bOpsStatusStop AND NOT(p_bBuffer1MagPresent OR p_bBuffer2MagPresent OR p_bBuffer3MagPresent);
//	ELSE
//		tyP0002Menu.tyMenu.tyBtnProdSel.uiMaskRtStat.0 	:= p_tyUsrMgmtCurrAccessRgt.bProdSel AND p_bOpsStatusStop AND NOT(p_bBuffer1MagPresent OR p_bBuffer2MagPresent);
//		tyP0002Menu.tyMenu.tyBtnMagSel.uiMaskRtStat.0	:= p_tyUsrMgmtCurrAccessRgt.bMagSel AND p_bOpsStatusStop AND NOT(p_bBuffer1MagPresent OR p_bBuffer2MagPresent);
//	END_IF

	IF p_tyNtParamCurr.eProjMag = ULMagTriple THEN
		tyP0002Menu.tyMenu.tyBtnProdSel.uiMaskRtStat.0 	:= p_bOpsStatusStop AND NOT(p_bBuffer1MagPresent OR p_bBuffer2MagPresent OR p_bBuffer3MagPresent);
		tyP0002Menu.tyMenu.tyBtnMagSel.uiMaskRtStat.0	:= p_bOpsStatusStop AND NOT(p_bBuffer1MagPresent OR p_bBuffer2MagPresent OR p_bBuffer3MagPresent);
	ELSE
		tyP0002Menu.tyMenu.tyBtnProdSel.uiMaskRtStat.0 	:= p_bOpsStatusStop AND NOT(p_bBuffer1MagPresent OR p_bBuffer2MagPresent);
		tyP0002Menu.tyMenu.tyBtnMagSel.uiMaskRtStat.0	:= p_bOpsStatusStop AND NOT(p_bBuffer1MagPresent OR p_bBuffer2MagPresent);
	END_IF

END_ACTION
```

#### Act_OptP0002ChgPage.st
```iecst
ACTION Act_OptP0002ChgPage:

	//General
	IF tyP0002Menu.tyMenu.tyBtnOpt.bRtCompl = TRUE THEN
		tyP0002Menu.tyMenu.tyBtnOpt.bRtCompl				:= FALSE;
		eChgPage											:= UIP0200OpsGen;

	ELSIF tyP0002Menu.tyMenu.tyBtnProdSel.bRtCompl = TRUE THEN
		tyP0002Menu.tyMenu.tyBtnProdSel.bRtCompl			:= FALSE;
		eChgPage											:= UIP0400ProdSel;

	ELSIF tyP0002Menu.tyMenu.tyBtnMagSel.bRtCompl = TRUE THEN
		tyP0002Menu.tyMenu.tyBtnMagSel.bRtCompl				:= FALSE;
		eChgPage											:= UIP0410MagSel;

	ELSIF tyP0002Menu.tyMenu.tyBtnMcInfo.bRtCompl = TRUE THEN
		tyP0002Menu.tyMenu.tyBtnMcInfo.bRtCompl				:= FALSE;
		eChgPage											:= UIP0300McInfo;

	ELSIF tyP0002Menu.tyMenu.tyBtnAlm.bRtCompl = TRUE THEN
		tyP0002Menu.tyMenu.tyBtnAlm.bRtCompl				:= FALSE;
		eChgPage											:= UIP0600Alm;

	ELSIF tyP0002Menu.tyMenu.tyBtnLogin.bRtCompl = TRUE THEN
		tyP0002Menu.tyMenu.tyBtnLogin.bRtCompl				:= FALSE;
		eChgPage											:= UIP0100Login;

	ELSIF tyP0002Menu.tyMenu.tyBtnLFCtrl.bRtCompl = TRUE THEN
		tyP0002Menu.tyMenu.tyBtnLFCtrl.bRtCompl				:= FALSE;
		eChgPage											:= UIP0700LFCtrl;

	ELSIF tyP0002Menu.tyMenu.tyBtnMagInfo.bRtCompl = TRUE THEN
		tyP0002Menu.tyMenu.tyBtnMagInfo.bRtCompl			:= FALSE;
		eChgPage											:= UIP0800MagInfo;

	ELSIF tyP0002Menu.tyMenu.tyBtnOvenInfo.bRtCompl = TRUE THEN
		tyP0002Menu.tyMenu.tyBtnOvenInfo.bRtCompl			:= FALSE;
		eChgPage											:= UIP0850OvenInfo;

	//Manual
	ELSIF tyP0002Menu.tyMenu.tyBtnGenInput.bRtCompl = TRUE THEN
		bUIManualMod										:= TRUE;
		tyP0002Menu.tyMenu.tyBtnGenInput.bRtCompl			:= FALSE;
		eChgPage											:= UIP0900GenIn;

	ELSIF tyP0002Menu.tyMenu.tyBtnGenOutput.bRtCompl = TRUE THEN
		bUIManualMod										:= TRUE;
		tyP0002Menu.tyMenu.tyBtnGenOutput.bRtCompl			:= FALSE;
		eChgPage											:= UIP0910GenOut;

	ELSIF tyP0002Menu.tyMenu.tyBtnMovCtrl.bRtCompl = TRUE THEN
		bUIManualMod										:= TRUE;
		tyP0002Menu.tyMenu.tyBtnMovCtrl.bRtCompl			:= FALSE;
		eChgPage											:= UIP0920MtrNPneuCtrl;

	ELSIF tyP0002Menu.tyMenu.tyBtnCommCtrl.bRtCompl = TRUE THEN
		bUIManualMod										:= TRUE;
		tyP0002Menu.tyMenu.tyBtnCommCtrl.bRtCompl			:= FALSE;
		eChgPage											:= UIP0940CommCtrl;

	ELSIF tyP0002Menu.tyMenu.tyBtnSimu.bRtCompl = TRUE THEN
		tyP0002Menu.tyMenu.tyBtnSimu.bRtCompl				:= FALSE;
		eChgPage											:= UIP0950Simu;

	//Settings
	ELSIF tyP0002Menu.tyMenu.tyBtnLang.bRtCompl = TRUE THEN
		tyP0002Menu.tyMenu.tyBtnLang.bRtCompl				:= FALSE;
		eChgPage											:= UIP1000Lang;

	ELSIF tyP0002Menu.tyMenu.tyBtnMcSet.bRtCompl = TRUE THEN
		tyP0002Menu.tyMenu.tyBtnMcSet.bRtCompl				:= FALSE;
		eChgPage											:= UIP1020McSetNavi;

	ELSIF tyP0002Menu.tyMenu.tyBtnMagSet.bRtCompl = TRUE THEN
		tyP0002Menu.tyMenu.tyBtnMagSet.bRtCompl				:= FALSE;
		eChgPage											:= UIP1030MagSet;

	ELSIF tyP0002Menu.tyMenu.tyBtnProdSet.bRtCompl = TRUE THEN
		tyP0002Menu.tyMenu.tyBtnProdSet.bRtCompl			:= FALSE;
		eChgPage											:= UIP1040ProdSet;

	ELSIF tyP0002Menu.tyMenu.tyBtnLFSet.bRtCompl = TRUE THEN
		tyP0002Menu.tyMenu.tyBtnLFSet.bRtCompl				:= FALSE;
		eChgPage											:= UIP1050LFSet;

	ELSIF tyP0002Menu.tyMenu.tyBtnUsrMgmt.bRtCompl = TRUE THEN
		tyP0002Menu.tyMenu.tyBtnUsrMgmt.bRtCompl			:= FALSE;
		eChgPage											:= UIP1080UsrMgmt;

	END_IF
	fbActSimuTmr (IN:= tyP0002Menu.tyMenu.tyBtnHotspotActSimu.bValue = TRUE ,PT:=T#8s);
	IF fbActSimuTmr.Q THEN
		IF tyP0002Menu.tyMenu.tyBtnSimu.uiRtStat =0 THEN
			tyP0002Menu.tyMenu.tyBtnSimu.uiRtStat := 1;
			fbActSimuTmr (IN:= FALSE);
		ELSE
			tyP0002Menu.tyMenu.tyBtnSimu.uiRtStat := 0;
			fbActSimuTmr (IN:= FALSE);
		END_IF
	END_IF
END_ACTION
```

#### Act_OptP0002ManualCtrl.st
```iecst
ACTION Act_OptP0002ManualCtrl:

	IF EDGEPOS(bUIManualMod) THEN

		tyP0910GenOut.tyGenOut.tyBtnTLAmber.bValue	:= TRUE;

		//Mask
		fUIInRtStatOff(ADR(tyP0002Menu.tyMenu.tyBitmapGen.uiMaskRtStat));
		fUIInRtStatOff(ADR(tyP0002Menu.tyMenu.tyBitmapSet.uiMaskRtStat));

		//Show Reset Manual Button
		fUIInRtStatOff(ADR(tyP0002Menu.tyMenu.tyBtnMnlRst.uiRtStat));

	END_IF

	IF tyP0002Menu.tyMenu.tyBtnMnlRst.bRtCompl = TRUE THEN
		tyP0002Menu.tyMenu.tyBtnMnlRst.bRtCompl	:= FALSE;

		bUIManualMod	:= FALSE;

		//Unmask
		fUIInRtStatHide(ADR(tyP0002Menu.tyMenu.tyBitmapGen.uiMaskRtStat));
		fUIInRtStatHide(ADR(tyP0002Menu.tyMenu.tyBitmapSet.uiMaskRtStat));

		//Hide Reset Manual Button
		fUIInRtStatHide(ADR(tyP0002Menu.tyMenu.tyBtnMnlRst.uiRtStat));

	END_IF

	bManualMod	:= bUIManualMod AND p_tyDI.bSafetyRlySig;

END_ACTION
```

#### Act_OptP0002MsgGuide.st
```iecst
ACTION Act_OptP0002MsgGuide:

	//Display
	tyP0002Menu.tyMenu.tyHotspotProdSel.uiRtStat.0	:= tyP0002Menu.tyMenu.tyBtnProdSel.uiMaskRtStat.0;
	tyP0002Menu.tyMenu.tyHotspotMagSel.uiRtStat.0	:= tyP0002Menu.tyMenu.tyBtnMagSel.uiMaskRtStat.0;

	IF p_tyNtParamCurr.eProjMag = ULMagTriple THEN
		tyP0002Menu.tyMenu.tyHotspotProdSel.bRtLk	:= NOT(p_bBuffer1MagPresent OR p_bBuffer2MagPresent OR p_bBuffer3MagPresent);
		tyP0002Menu.tyMenu.tyHotspotMagSel.bRtLk	:= NOT(p_bBuffer1MagPresent OR p_bBuffer2MagPresent OR p_bBuffer3MagPresent);
	ELSE
		tyP0002Menu.tyMenu.tyHotspotProdSel.bRtLk	:= NOT(p_bBuffer1MagPresent OR p_bBuffer2MagPresent);
		tyP0002Menu.tyMenu.tyHotspotMagSel.bRtLk	:= NOT(p_bBuffer1MagPresent OR p_bBuffer2MagPresent);
	END_IF

	//Control
	IF tyP0002Menu.tyMenu.tyHotspotProdSel.bRtCompl OR tyP0002Menu.tyMenu.tyHotspotMagSel.bRtCompl THEN
		p_tyC0008MsgBox ACCESS ADR(tyP0002Menu.tyMsgBoxRemoveMag);

		IF tyP0002Menu.tyMsgBoxRemoveMag.tyBtnNo.bRtCompl = TRUE THEN
			tyP0002Menu.tyMsgBoxRemoveMag.tyBtnNo.bRtCompl	:= FALSE;
			tyP0002Menu.tyMsgBoxRemoveMag.tyBtnNo.bValue	:= FALSE;

			p_tyC0008MsgBox ACCESS ADR(tyP0002Menu.tyMsgBoxHide);

			IF tyP0002Menu.tyMenu.tyHotspotProdSel.bRtCompl AND tyP0002Menu.tyMenu.tyBtnProdSel.uiMaskRtStat.0 THEN
				eChgPage	:= UIP0400ProdSel;

			ELSIF tyP0002Menu.tyMenu.tyHotspotMagSel.bRtCompl AND tyP0002Menu.tyMenu.tyBtnMagSel.uiMaskRtStat.0 THEN
				eChgPage	:= UIP0410MagSel;

			END_IF

			tyP0002Menu.tyMenu.tyHotspotProdSel.bRtCompl	:= FALSE;
			tyP0002Menu.tyMenu.tyHotspotMagSel.bRtCompl		:= FALSE;

		END_IF

	END_IF

END_ACTION
```

#### Act_OptP0002UpdtData.st
```iecst
ACTION Act_OptP0002UpdtData:

	IF bLoginSuccess = FALSE THEN
		tyP0002Menu.tyMenu.tyBtnLogin.usiBitmapIdx		:= 0;
		tyP0002Menu.tyMenu.tyBtnLogin.usiTxtIdx			:= 0;
	ELSE
		tyP0002Menu.tyMenu.tyBtnLogin.usiBitmapIdx		:= 1;
		tyP0002Menu.tyMenu.tyBtnLogin.usiTxtIdx			:= 1;
	END_IF

	tyP0100Login.tyLogin.tyBtnLogin.bRtCompl := FALSE;

END_ACTION
```

#### Act_EntP0003Disp.st
```iecst
ACTION Act_EntP0003Disp:

	//Access
	p_tyC0005Main ACCESS ADR(tyCommon.tyMain1);

	p_tyC0007Notif ACCESS ADR(tyCommon.tyNotif);

	p_tyP0003Gen ACCESS ADR(tyP0003MMenu.tyMMenuGen);

	IF NOT bPromptSessionExp THEN
		p_tyC0008MsgBox ACCESS ADR(tyP0003MMenu.tyMsgBoxHide);
	END_IF

	p_tyC0009Info ACCESS ADR(tyCommon.tyInfo);

	p_tyP0003BtnAuto ACCESS ADR(tyP0003MMenu.tyMMenuBtn.tyBtnAuto);
	p_tyP0003BtnStop ACCESS ADR(tyP0003MMenu.tyMMenuBtn.tyBtnStop);
	p_tyP0003BtnReset ACCESS ADR(tyP0003MMenu.tyMMenuBtn.tyBtnReset);
	p_tyP0003BtnBuz ACCESS ADR(tyP0003MMenu.tyMMenuBtn.tyBtnBuz);
	p_tyP0003AcceptData ACCESS ADR(tyP0003MMenu.tyMMenuBtn.tyBtnAccDat);

	//Communication
	tyP0200OpsGen.tyUSCommB.tyLyr.uiRtStat.0 := NOT(p_tyNtParamCurr.bProjLaneBPrep);
	//hide corresponding button
	tyP0003MMenu.tyMMenuBtn.tyBtnRlsNewMag1.uiRtStat.0 := p_tyMcParamCurr.eMagExMode = McSetMagXcAutoMode AND p_tyMcParamCurr.eAGVComProtocol <> McSetAGVCommDisabled OR p_tyNtParamCurr.bProjLifterMagPlatform;
	tyP0003MMenu.tyMMenuBtn.tyBtnRlsNewMag2.uiRtStat.0 := p_tyMcParamCurr.eMagExMode = McSetMagXcAutoMode AND p_tyMcParamCurr.eAGVComProtocol <> McSetAGVCommDisabled OR p_tyNtParamCurr.bProjLifterMagPlatform;
	tyP0003MMenu.tyMMenuBtn.tyBtnRlsNewMag3.uiRtStat.0 := p_tyMcParamCurr.eMagExMode = McSetMagXcAutoMode AND p_tyMcParamCurr.eAGVComProtocol <> McSetAGVCommDisabled OR p_tyNtParamCurr.bProjLifterMagPlatform;

	//Occupied
	usiPosidx := 0 ;
	FOR usidx:= 1 TO SIZEOF(p_tyMcParamCurr.tyOptBtnPos)/SIZEOF(p_tyMcParamCurr.tyOptBtnPos.ePos1) DO
		IF NOT(p_tyNtParamCurr.tyDOSettings.diBuzzer > 0 AND usidx = 1)THEN

			p_eCurrBtnPos ACCESS (ADR(p_tyMcParamCurr.tyOptBtnPos) + (usiPosidx)*SIZEOF(p_tyMcParamCurr.tyOptBtnPos.ePos1));

			IF p_eCurrBtnPos = eNA THEN
				a_tyPtrtoAddr[usidx] :=   ADR(tyP0003MMenu.tyMMenuBtn.tyBtnHide);
			ELSIF p_eCurrBtnPos = eMagUnload THEN
				a_tyPtrtoAddr[usidx] :=   ADR(tyP0003MMenu.tyMMenuBtn.tyBtnMnlUnload);
			ELSIF p_eCurrBtnPos= eRlsNewMagazine1 THEN
				a_tyPtrtoAddr[usidx] :=   ADR(tyP0003MMenu.tyMMenuBtn.tyBtnRlsNewMag1);
			ELSIF p_eCurrBtnPos= eRlsNewMagazine2 THEN
				a_tyPtrtoAddr[usidx] :=   ADR(tyP0003MMenu.tyMMenuBtn.tyBtnRlsNewMag2);
			ELSIF p_eCurrBtnPos = eRlsNewMagazine3 THEN
				a_tyPtrtoAddr[usidx] :=   ADR(tyP0003MMenu.tyMMenuBtn.tyBtnRlsNewMag3);
			END_IF
			usiPosidx := usiPosidx +1;
		ELSE
			a_tyPtrtoAddr[usidx] :=   ADR(tyP0003MMenu.tyMMenuBtn.tyBtnHide);
		END_IF
	END_FOR
	p_tyP0003Btn1 ACCESS a_tyPtrtoAddr[1];
	p_tyP0003Btn2 ACCESS a_tyPtrtoAddr[2];
	p_tyP0003Btn3 ACCESS a_tyPtrtoAddr[3];
	p_tyP0003Btn4 ACCESS a_tyPtrtoAddr[4];
	p_tyP0003Btn5 ACCESS a_tyPtrtoAddr[5];
	p_tyP0003Btn6 ACCESS a_tyPtrtoAddr[6];
	p_tyP0003Btn7 ACCESS a_tyPtrtoAddr[7];

	//Not Used
//	p_tyP0003Btn4 ACCESS ADR(tyP0003MMenu.tyMMenuBtn.tyBtn4);// If not used, hide it in the data type
//	p_tyP0003Btn5 ACCESS ADR(tyP0003MMenu.tyMMenuBtn.tyBtn5);// If not used, hide it in the data type
//	p_tyP0003Btn6 ACCESS ADR(tyP0003MMenu.tyMMenuBtn.tyBtn6);// If not used, hide it in the data type
//    p_tyP0003Btn7 ACCESS ADR(tyP0003MMenu.tyMMenuBtn.tyBtn7);// If not used, hide it in the data type

END_ACTION
```

#### Act_OptP0003UpdtStat.st
```iecst
ACTION Act_OptP0003UpdtStat:

	IF p_bOpsStatusRun THEN
		tyP0003MMenu.tyMMenuGen.tyStatusTxt.usiValueIdx := 20;
	ELSIF p_bOpsStatusCycleStop THEN
		tyP0003MMenu.tyMMenuGen.tyStatusTxt.usiValueIdx := 21;
	ELSIF p_bAlarmErr THEN
		tyP0003MMenu.tyMMenuGen.tyStatusTxt.usiValueIdx := 22;
	ELSE
		tyP0003MMenu.tyMMenuGen.tyStatusTxt.usiValueIdx := 23;
	END_IF

	//SMEMA Indicator
	IF p_tyNtParamCurr.bUIConvDirRL = FALSE THEN
		fUIInRtStatHide(ADR(tyP0003MMenu.tyMMenuGen.tyBitmapUSAComm1.uiMaskRtStat));
		fUIInRtStatHide(ADR(tyP0003MMenu.tyMMenuGen.tyBitmapUSBComm1.uiMaskRtStat));
		IF p_tyMcParamCurr.eUSCommA = McSetCommModSMEMA THEN
			fUIInRtStatHide(ADR(tyP0003MMenu.tyMMenuGen.tyBitmapUSAComm.uiMaskRtStat));
		ELSIF p_tyMcParamCurr.eUSCommA = McSetCommModHermes THEN
			IF p_bUSHermesAConnected = TRUE THEN
				fUIInRtStatHide(ADR(tyP0003MMenu.tyMMenuGen.tyBitmapUSAComm.uiMaskRtStat));
			ELSE
				fUIInRtStatOff(ADR(tyP0003MMenu.tyMMenuGen.tyBitmapUSAComm.uiMaskRtStat));
			END_IF
		END_IF

		IF p_tyMcParamCurr.eUSCommB = McSetCommModSMEMA THEN
			fUIInRtStatHide(ADR(tyP0003MMenu.tyMMenuGen.tyBitmapUSBComm.uiMaskRtStat));
		ELSIF p_tyMcParamCurr.eUSCommB = McSetCommModHermes THEN
			IF p_bUSHermesBConnected = TRUE THEN
				fUIInRtStatHide(ADR(tyP0003MMenu.tyMMenuGen.tyBitmapUSBComm.uiMaskRtStat));
			ELSE
				fUIInRtStatOff(ADR(tyP0003MMenu.tyMMenuGen.tyBitmapUSBComm.uiMaskRtStat));
			END_IF
		END_IF
	ELSE
		fUIInRtStatHide(ADR(tyP0003MMenu.tyMMenuGen.tyBitmapUSAComm.uiMaskRtStat));
		fUIInRtStatHide(ADR(tyP0003MMenu.tyMMenuGen.tyBitmapUSBComm.uiMaskRtStat));
		IF p_tyMcParamCurr.eUSCommA = McSetCommModSMEMA THEN
			fUIInRtStatHide(ADR(tyP0003MMenu.tyMMenuGen.tyBitmapUSAComm1.uiMaskRtStat));
		ELSIF p_tyMcParamCurr.eUSCommA = McSetCommModHermes THEN
			IF p_bUSHermesAConnected = TRUE THEN
				fUIInRtStatHide(ADR(tyP0003MMenu.tyMMenuGen.tyBitmapUSAComm1.uiMaskRtStat));
			ELSE
				fUIInRtStatOff(ADR(tyP0003MMenu.tyMMenuGen.tyBitmapUSAComm1.uiMaskRtStat));
			END_IF
		END_IF

		IF p_tyMcParamCurr.eUSCommB = McSetCommModSMEMA THEN
			fUIInRtStatHide(ADR(tyP0003MMenu.tyMMenuGen.tyBitmapUSBComm1.uiMaskRtStat));
		ELSIF p_tyMcParamCurr.eUSCommB = McSetCommModHermes THEN
			IF p_bUSHermesBConnected = TRUE THEN
				fUIInRtStatHide(ADR(tyP0003MMenu.tyMMenuGen.tyBitmapUSBComm1.uiMaskRtStat));
			ELSE
				fUIInRtStatOff(ADR(tyP0003MMenu.tyMMenuGen.tyBitmapUSBComm1.uiMaskRtStat));
			END_IF
		END_IF
	END_IF
	//USB A
	IF p_tyMcParamCurr.eUSCommA = McSetCommModSMEMA THEN
		IF p_tyNtParamCurr.bUIConvDirRL = FALSE THEN

			IF p_bUSSMEMAADSRdy = TRUE THEN
				tyP0003MMenu.tyMMenuGen.tyBitmapUSOut.usiValueIdx	:= 1;
			ELSE
				tyP0003MMenu.tyMMenuGen.tyBitmapUSOut.usiValueIdx	:= 0;
			END_IF
		ELSE
			IF p_bUSSMEMAADSRdy = TRUE THEN
				tyP0003MMenu.tyMMenuGen.tyBitmapUSOut1.usiValueIdx	:= 1;
			ELSE
				tyP0003MMenu.tyMMenuGen.tyBitmapUSOut1.usiValueIdx	:= 0;
			END_IF
		END_IF

	ELSIF p_tyMcParamCurr.eUSCommA = McSetCommModHermes THEN
		IF p_tyNtParamCurr.bUIConvDirRL = FALSE THEN
			IF p_bUSHermesADSRdy = TRUE THEN
				IF p_bUSHermesADSGdRdy = TRUE THEN
					tyP0003MMenu.tyMMenuGen.tyBitmapUSOut.usiValueIdx	:= 1;
				ELSE
					tyP0003MMenu.tyMMenuGen.tyBitmapUSOut.usiValueIdx	:= 2;
				END_IF
			ELSE
				tyP0003MMenu.tyMMenuGen.tyBitmapUSOut.usiValueIdx		:= 0;
			END_IF
		ELSE
			IF p_bUSHermesADSRdy = TRUE THEN
				IF p_bUSHermesADSGdRdy = TRUE THEN
					tyP0003MMenu.tyMMenuGen.tyBitmapUSOut1.usiValueIdx	:= 1;
				ELSE
					tyP0003MMenu.tyMMenuGen.tyBitmapUSOut1.usiValueIdx	:= 2;
				END_IF
			ELSE
				tyP0003MMenu.tyMMenuGen.tyBitmapUSOut1.usiValueIdx		:= 0;
			END_IF
		END_IF

	END_IF

	//UBA A
	IF p_tyMcParamCurr.eUSCommA = McSetCommModSMEMA THEN

		IF p_tyNtParamCurr.bUIConvDirRL = FALSE THEN
			IF p_bUSSMEMAAUSRdy = TRUE THEN
				IF p_bUSSMEMAAUSGdBrdRdy = TRUE THEN
					tyP0003MMenu.tyMMenuGen.tyBitmapUSIn.usiValueIdx	:= 1;
				ELSE
					tyP0003MMenu.tyMMenuGen.tyBitmapUSIn.usiValueIdx	:= 2;
				END_IF
			ELSE
				tyP0003MMenu.tyMMenuGen.tyBitmapUSIn.usiValueIdx		:= 0;
			END_IF
		ELSE
			IF p_bUSSMEMAAUSRdy = TRUE THEN
				IF p_bUSSMEMAAUSGdBrdRdy = TRUE THEN
					tyP0003MMenu.tyMMenuGen.tyBitmapUSIn1.usiValueIdx	:= 1;
				ELSE
					tyP0003MMenu.tyMMenuGen.tyBitmapUSIn1.usiValueIdx	:= 2;
				END_IF
			ELSE
				tyP0003MMenu.tyMMenuGen.tyBitmapUSIn1.usiValueIdx		:= 0;
			END_IF
		END_IF

	ELSIF p_tyMcParamCurr.eUSCommA = McSetCommModHermes THEN

		IF p_tyNtParamCurr.bUIConvDirRL = FALSE THEN
			IF p_bUSHermesAUSRdy = TRUE THEN
				IF p_bUSHermesAUSGdRdy = TRUE THEN
					tyP0003MMenu.tyMMenuGen.tyBitmapUSIn.usiValueIdx	:= 1;
				ELSE
					tyP0003MMenu.tyMMenuGen.tyBitmapUSIn.usiValueIdx	:= 2;
				END_IF
			ELSE
				tyP0003MMenu.tyMMenuGen.tyBitmapUSIn.usiValueIdx		:= 0;
			END_IF
		ELSE
			IF p_bUSHermesAUSRdy = TRUE THEN
				IF p_bUSHermesAUSGdRdy = TRUE THEN
					tyP0003MMenu.tyMMenuGen.tyBitmapUSIn1.usiValueIdx	:= 1;
				ELSE
					tyP0003MMenu.tyMMenuGen.tyBitmapUSIn1.usiValueIdx	:= 2;
				END_IF
			ELSE
				tyP0003MMenu.tyMMenuGen.tyBitmapUSIn1.usiValueIdx		:= 0;
			END_IF
		END_IF

	END_IF

	//USB B
	IF p_tyMcParamCurr.eUSCommB = McSetCommModSMEMA THEN
		IF p_tyNtParamCurr.bUIConvDirRL = FALSE THEN

			IF p_bUSSMEMABDSRdy = TRUE THEN
				tyP0003MMenu.tyMMenuGen.tyBitmapUSBOut.usiValueIdx	:= 1;
			ELSE
				tyP0003MMenu.tyMMenuGen.tyBitmapUSBOut.usiValueIdx	:= 0;
			END_IF

		ELSE

			IF p_bUSSMEMABDSRdy = TRUE THEN
				tyP0003MMenu.tyMMenuGen.tyBitmapUSBOut1.usiValueIdx	:= 1;
			ELSE
				tyP0003MMenu.tyMMenuGen.tyBitmapUSBOut1.usiValueIdx	:= 0;
			END_IF

		END_IF

	ELSIF p_tyMcParamCurr.eUSCommB = McSetCommModHermes THEN

		IF p_tyNtParamCurr.bUIConvDirRL THEN
			IF p_bUSHermesBDSRdy = TRUE THEN
				IF p_bUSHermesBDSGdRdy = TRUE THEN
					tyP0003MMenu.tyMMenuGen.tyBitmapUSBOut.usiValueIdx	:= 1;
				ELSE
					tyP0003MMenu.tyMMenuGen.tyBitmapUSBOut.usiValueIdx	:= 2;
				END_IF
			ELSE
				tyP0003MMenu.tyMMenuGen.tyBitmapUSBOut.usiValueIdx		:= 0;
			END_IF
		ELSE
			IF p_bUSHermesBDSRdy = TRUE THEN
				IF p_bUSHermesBDSGdRdy = TRUE THEN
					tyP0003MMenu.tyMMenuGen.tyBitmapUSBOut1.usiValueIdx	:= 1;
				ELSE
					tyP0003MMenu.tyMMenuGen.tyBitmapUSBOut1.usiValueIdx	:= 2;
				END_IF
			ELSE
				tyP0003MMenu.tyMMenuGen.tyBitmapUSBOut1.usiValueIdx		:= 0;
			END_IF
		END_IF

	END_IF

	//UBA B
	IF p_tyMcParamCurr.eUSCommB = McSetCommModSMEMA THEN

		IF p_tyNtParamCurr.bUIConvDirRL = FALSE THEN
			IF p_bUSSMEMABUSRdy = TRUE THEN
				IF p_bUSSMEMABUSGdBrdRdy = TRUE THEN
					tyP0003MMenu.tyMMenuGen.tyBitmapUSBIn.usiValueIdx	:= 1;
				ELSE
					tyP0003MMenu.tyMMenuGen.tyBitmapUSBIn.usiValueIdx	:= 2;
				END_IF
			ELSE
				tyP0003MMenu.tyMMenuGen.tyBitmapUSBIn.usiValueIdx		:= 0;
			END_IF
		ELSE
			IF p_bUSSMEMABUSRdy = TRUE THEN
				IF p_bUSSMEMABUSGdBrdRdy = TRUE THEN
					tyP0003MMenu.tyMMenuGen.tyBitmapUSBIn1.usiValueIdx	:= 1;
				ELSE
					tyP0003MMenu.tyMMenuGen.tyBitmapUSBIn1.usiValueIdx	:= 2;
				END_IF
			ELSE
				tyP0003MMenu.tyMMenuGen.tyBitmapUSBIn1.usiValueIdx		:= 0;
			END_IF
		END_IF

	ELSIF p_tyMcParamCurr.eUSCommB = McSetCommModHermes THEN

		IF p_tyNtParamCurr.bUIConvDirRL = FALSE THEN
			IF p_bUSHermesBUSRdy = TRUE THEN
				IF p_bUSHermesBUSGdRdy = TRUE THEN
					tyP0003MMenu.tyMMenuGen.tyBitmapUSBIn.usiValueIdx	:= 1;
				ELSE
					tyP0003MMenu.tyMMenuGen.tyBitmapUSBIn.usiValueIdx	:= 2;
				END_IF
			ELSE
				tyP0003MMenu.tyMMenuGen.tyBitmapUSBIn.usiValueIdx		:= 0;
			END_IF
		ELSE
			IF p_bUSHermesBUSRdy = TRUE THEN
				IF p_bUSHermesBUSGdRdy = TRUE THEN
					tyP0003MMenu.tyMMenuGen.tyBitmapUSBIn1.usiValueIdx	:= 1;
				ELSE
					tyP0003MMenu.tyMMenuGen.tyBitmapUSBIn1.usiValueIdx	:= 2;
				END_IF
			ELSE
				tyP0003MMenu.tyMMenuGen.tyBitmapUSBIn1.usiValueIdx		:= 0;
			END_IF
		END_IF

	END_IF

	//Current last zone product recipe name

	tyP0003MMenu.tyMMenuGen.tyStringProdNm.sValue := p_tyProdRcpCurrRcp1.sRcpNm;

END_ACTION
```

#### Act_EntP0100Disp.st
```iecst
ACTION Act_EntP0100Disp:

	//Access Address
	p_tyC0005Main ACCESS ADR(tyCommon.tyMain);

	p_tyC0007Notif ACCESS ADR(tyCommon.tyNotif);

	p_tyC0008MsgBox ACCESS ADR(tyP0100Login.tyMsgBoxHide);

	p_tyC0009Info ACCESS ADR(tyCommon.tyInfo);

	p_tyP0100Login ACCESS ADR(tyP0100Login.tyLogin);

	p_tyP0100Logout ACCESS ADR(tyP0100Login.tyLogout);

	//Clear Input
	tyP0100Login.tyLogin.tyStringUsrNm.sValue	:= '';
	tyP0100Login.tyLogin.tyStringPw.sValue		:= '';

	//Login Logout Layer
	IF  bLoginSuccess = TRUE THEN
		fUIInRtStatOff(ADR(tyP0100Login.tyLogout.tyLyr.uiRtStat));
		fUIInRtStatHide(ADR(tyP0100Login.tyLogin.tyLyr.uiRtStat));
	ELSE
		fUIInRtStatHide(ADR(tyP0100Login.tyLogout.tyLyr.uiRtStat));
		fUIInRtStatOff(ADR(tyP0100Login.tyLogin.tyLyr.uiRtStat));
	END_IF

	//Bypass Hotspot
	IF p_tyUsrMgmtAdminList[1].sUsrNm = '' THEN
		fUIInRtStatOff(ADR(tyP0100Login.tyLogin.tyHotspotBypassLogin.uiRtStat));
	ELSE
		fUIInRtStatHide(ADR(tyP0100Login.tyLogin.tyHotspotBypassLogin.uiRtStat));
	END_IF

	//Reset User Level Hotspot
	tyP0100Login.tyLogin.tyBtnLogin.usiBitmapIdx	:= 0;

END_ACTION
```

#### Act_OptP0100NomLogin.st
```iecst
ACTION Act_OptP0100NomLogin:

	IF tyP0100Login.tyLogin.tyBtnLogin.bRtCompl = TRUE THEN

		IF usiLoginStep = 0 THEN
			tyUsrMgmtInfoIn.sUsrNm := tyP0100Login.tyLogin.tyStringUsrNm.sValue;
			tyUsrMgmtInfoIn.sPw := tyP0100Login.tyLogin.tyStringPw.sValue;

			usiLoginStep := 1;

		ELSIF usiLoginStep = 1 THEN
			//User Login
			eUsrMgmtAct := UsrMgmtActLogin;

			IF p_eUsrMgmtStat = UsrMgmtActLogin AND p_eUsrMgmtStatus = Done THEN
				eUsrMgmtAct := UsrMgmtActIdle;

				IF p_bUsrMgmtNmNotExist = TRUE THEN
					usiLoginStep := 2;
				ELSE
					IF p_bUsrMgmtLoginSuccess = TRUE AND p_bUsrMgmtPwMismatch = FALSE THEN
						usiLoginStep := 3;
					ELSIF p_bUsrMgmtLoginSuccess = FALSE AND p_bUsrMgmtPwMismatch = TRUE THEN
						usiLoginStep := 4;
					END_IF
				END_IF

			END_IF

		ELSIF usiLoginStep = 2 THEN
			//Name Not Exist
			p_tyC0008MsgBox ACCESS ADR(tyP0100Login.tyMsgBoxNmNotExist);

			IF tyP0100Login.tyMsgBoxNmNotExist.tyBtnNo.bRtCompl = TRUE THEN
				tyP0100Login.tyMsgBoxNmNotExist.tyBtnNo.bRtCompl := FALSE;
				tyP0100Login.tyMsgBoxNmNotExist.tyBtnNo.bValue := FALSE;

				p_tyC0008MsgBox ACCESS ADR(tyP0100Login.tyMsgBoxHide);

				usiLoginStep := 97;
			END_IF

		ELSIF usiLoginStep = 3 THEN
			//User Login Success
			tyP1080UsrMgmt.tyUsrMgmt.tyDrpDnLvl.usiValueMinIdx := 0;
			tyP1080UsrMgmt.tyUsrMgmt.tyDrpDnLvl.usiValueMaxIdx := 3;

			tyP1080UsrMgmt.tyCreate.tyDrpDnLvl.usiValueMinIdx := 0;
			tyP1080UsrMgmt.tyCreate.tyDrpDnLvl.usiValueMaxIdx := 2;

			tyP1080UsrMgmt.tyEdit.tyDrpDnLvl.usiValueMinIdx := 0;
			tyP1080UsrMgmt.tyEdit.tyDrpDnLvl.usiValueMaxIdx := 2;

			usiLoginStep := 99;

		ELSIF usiLoginStep = 4 THEN
			//Password Mismatch
			p_tyC0008MsgBox ACCESS ADR(tyP0100Login.tyMsgBoxPwMismatch);

			IF tyP0100Login.tyMsgBoxPwMismatch.tyBtnNo.bRtCompl = TRUE THEN
				tyP0100Login.tyMsgBoxPwMismatch.tyBtnNo.bRtCompl := FALSE;
				tyP0100Login.tyMsgBoxPwMismatch.tyBtnNo.bValue := FALSE;

				p_tyC0008MsgBox ACCESS ADR(tyP0100Login.tyMsgBoxHide);

				usiLoginStep := 98;
			END_IF

		ELSIF usiLoginStep = 97 THEN
			tyP0100Login.tyLogin.tyStringUsrNm.sValue := '';
			tyP0100Login.tyLogin.tyStringPw.sValue := '';

			tyP0100Login.tyLogin.tyBtnLogin.bRtCompl := FALSE;
			tyP0100Login.tyLogin.tyBtnLogin.bValue := FALSE;

			usiLoginStep := 0;

		ELSIF usiLoginStep = 98 THEN
			tyP0100Login.tyLogin.tyStringPw.sValue := '';

			tyP0100Login.tyLogin.tyBtnLogin.bRtCompl := FALSE;
			tyP0100Login.tyLogin.tyBtnLogin.bValue := FALSE;

			usiLoginStep := 0;

		ELSIF usiLoginStep = 99 THEN
			eChgPage := UIP0002Menu;
			bLoginSuccess := TRUE;

			tyP0100Login.tyLogin.tyStringUsrNm.sValue := '';
			tyP0100Login.tyLogin.tyStringPw.sValue := '';

			tyP0100Login.tyLogin.tyBtnLogin.bRtCompl := FALSE;
			tyP0100Login.tyLogin.tyBtnLogin.bValue := FALSE;

			usiLoginStep := 0;

		END_IF

	END_IF

END_ACTION
```

#### Act_OptP0100BypassLogin.st
```iecst
ACTION Act_OptP0100BypassLogin:

	IF tyP0100Login.tyLogin.tyHotspotBypassLogin.bRtCompl = TRUE THEN

		IF (tyP0100Login.tyLogin.tyStringUsrNm.sValue = p_tyNtParamCurr.sUIDefaultLoginNm) AND (tyP0100Login.tyLogin.tyStringPw.sValue = p_tyNtParamCurr.sUIDefaultLoginPw) THEN

			eUsrMgmtAct := UsrMgmtActBypassLogin;

			IF p_eUsrMgmtStat = UsrMgmtActBypassLogin AND p_eUsrMgmtStatus = Done THEN
				eUsrMgmtAct		:= UsrMgmtActIdle;
				bLoginSuccess	:= TRUE;

				//Update
				tyP1080UsrMgmt.tyUsrMgmt.tyDrpDnLvl.usiValueMinIdx	:= 0;
				tyP1080UsrMgmt.tyUsrMgmt.tyDrpDnLvl.usiValueMaxIdx	:= 3;

				tyP1080UsrMgmt.tyCreate.tyDrpDnLvl.usiValueMinIdx	:= 0;
				tyP1080UsrMgmt.tyCreate.tyDrpDnLvl.usiValueMaxIdx	:= 2;

				tyP1080UsrMgmt.tyEdit.tyDrpDnLvl.usiValueMinIdx		:= 0;
				tyP1080UsrMgmt.tyEdit.tyDrpDnLvl.usiValueMaxIdx		:= 2;

				eChgPage	:= UIP0002Menu;

				tyP0100Login.tyLogin.tyHotspotBypassLogin.bRtCompl	:= FALSE;
			END_IF

		ELSE

			p_tyC0008MsgBox ACCESS ADR(tyP0100Login.tyMsgBoxPwMismatch);

			IF tyP0100Login.tyMsgBoxPwMismatch.tyBtnNo.bRtCompl = TRUE THEN
				tyP0100Login.tyMsgBoxPwMismatch.tyBtnNo.bRtCompl	:= FALSE;
				tyP0100Login.tyMsgBoxPwMismatch.tyBtnNo.bValue		:= FALSE;

				p_tyC0008MsgBox ACCESS ADR(tyP0100Login.tyMsgBoxHide);

			//	tyP0100Login.tyLogin.tyStringUsrNm.sValue	:= '';
				tyP0100Login.tyLogin.tyStringPw.sValue		:= '';

				tyP0100Login.tyLogin.tyHotspotBypassLogin.bRtCompl	:= FALSE;
			END_IF

		END_IF

	END_IF

END_ACTION
```

#### Act_OptP0100Logout.st
```iecst
ACTION Act_OptP0100Logout:

	IF tyP0100Login.tyLogout.tyBtnLogout.bRtCompl THEN
		eUsrMgmtAct	:= UsrMgmtActLogout;

		IF p_eUsrMgmtStat = UsrMgmtActLogout AND p_eUsrMgmtStatus = Done THEN
			eUsrMgmtAct	:= UsrMgmtActIdle;

			bLoginSuccess	:= FALSE;

			//Update
			tyP0100Login.tyLogin.tyStringUsrNm.sValue	:= '';
			tyP0100Login.tyLogin.tyStringPw.sValue		:= '';

			tyP0100Login.tyLogout.tyBtnLogout.bRtCompl	:= FALSE;
			tyP0100Login.tyLogout.tyBtnLogout.bValue	:= FALSE;

			fUIInRtStatHide(ADR(tyP0100Login.tyLogout.tyLyr.uiRtStat));
			fUIInRtStatOff(ADR(tyP0100Login.tyLogin.tyLyr.uiRtStat));
		END_IF

	END_IF

END_ACTION
```

#### Act_OptP0100Keypad.st
```iecst
ACTION Act_OptP0100Keypad:

	IF fUIOutRtStatTPIsOpen(ADR(tyP0100Login.tyLogin.tyStringUsrNm.uiRtStat)) = TRUE THEN
		tyProperty.tyKeypad.tyStringTitle.sKeypadTitle	:= tyP0100Login.tyLogin.tyStringUsrNm.sKeypadTitle;

	ELSIF fUIOutRtStatTPIsOpen(ADR(tyP0100Login.tyLogin.tyStringPw.uiRtStat)) = TRUE THEN
		tyProperty.tyKeypad.tyStringTitle.sKeypadTitle	:= tyP0100Login.tyLogin.tyStringPw.sKeypadTitle;

	ELSE
		tyProperty.tyKeypad.tyStringTitle.sKeypadTitle	:= '';

	END_IF

END_ACTION
```
